gfCNCPoint5[2424] = {X 421.3630, Y 54.1078, Z -6.3333, A 0.000, B 0.000, C 0.000 }
gfCNCPoint5[2425] = {X 422.1821, Y 54.6225, Z -6.3333, A 0.000, B 0.000, C 0.000 }
gfCNCPoint5[2426] = {X 422.8661, Y 55.3065, Z -6.3333, A 0.000, B 0.000, C 0.000 }
gfCNCPoint5[2427] = {X 423.3808, Y 56.1256, Z -6.3333, A 0.000, B 0.000, C 0.000 }
gfCNCPoint5[2428] = {X 423.7003, Y 57.0387, Z -6.3333, A 0.000, B 0.000, C 0.000 }
gfCNCPoint5[2429] = {X 423.8086, Y 58.0000, Z -6.3333, A 0.000, B 0.000, C 0.000 }
gfCNCPoint5[2430] = {X 423.8086, Y 58.2318, Z -6.3333, A 0.000, B 0.000, C 0.000 }
gfCNCPoint5[2431] = {X 429.6116, Y 60.4927, Z -6.3333, A 0.000, B 0.000, C 0.000 }
gfCNCPoint5[2432] = {X 457.8582, Y 71.7001, Z -6.3333, A 0.000, B 0.000, C 0.000 }
gfCNCPoint5[2433] = {X 457.8604, Y 63.2123, Z -6.3333, A 0.000, B 0.000, C 0.000 }
gfCNCPoint5[2434] = {X 457.0088, Y 63.0032, Z -6.3333, A 0.000, B 0.000, C 0.000 }
gfCNCPoint5[2435] = {X 456.2169, Y 62.6263, Z -6.3333, A 0.000, B 0.000, C 0.000 }
gfCNCPoint5[2436] = {X 455.5175, Y 62.0974, Z -6.3333, A 0.000, B 0.000, C 0.000 }
gfCNCPoint5[2437] = {X 454.9393, Y 61.4381, Z -6.3333, A 0.000, B 0.000, C 0.000 }
gfCNCPoint5[2438] = {X 454.5062, Y 60.6756, Z -6.3333, A 0.000, B 0.000, C 0.000 }
gfCNCPoint5[2439] = {X 454.2360, Y 59.8414, Z -6.3333, A 0.000, B 0.000, C 0.000 }
gfCNCPoint5[2440] = {X 454.1398, Y 58.9697, Z -6.3333, A 0.000, B 0.000, C 0.000 }
gfCNCPoint5[2441] = {X 454.1396, Y 58.0000, Z -6.3333, A 0.000, B 0.000, C 0.000 }
gfCNCPoint5[2442] = {X 454.2479, Y 57.0387, Z -6.3333, A 0.000, B 0.000, C 0.000 }
gfCNCPoint5[2443] = {X 454.5674, Y 56.1256, Z -6.3333, A 0.000, B 0.000, C 0.000 }
gfCNCPoint5[2444] = {X 455.0821, Y 55.3065, Z -6.3333, A 0.000, B 0.000, C 0.000 }
gfCNCPoint5[2445] = {X 455.7661, Y 54.6225, Z -6.3333, A 0.000, B 0.000, C 0.000 }
gfCNCPoint5[2446] = {X 456.5852, Y 54.1078, Z -6.3333, A 0.000, B 0.000, C 0.000 }
gfCNCPoint5[2447] = {X 457.4983, Y 53.7883, Z -6.3333, A 0.000, B 0.000, C 0.000 }
gfCNCPoint5[2448] = {X 458.4596, Y 53.6800, Z -6.3333, A 0.000, B 0.000, C 0.000 }
gfCNCPoint5[2449] = {X 475.0000, Y 53.6800, Z -6.3333, A 0.000, B 0.000, C 0.000 }
gfCNCPoint5[2450] = {X 475.9613, Y 53.7883, Z -6.3333, A 0.000, B 0.000, C 0.000 }
gfCNCPoint5[2451] = {X 476.8744, Y 54.1078, Z -6.3333, A 0.000, B 0.000, C 0.000 }
gfCNCPoint5[2452] = {X 477.6935, Y 54.6225, Z -6.3333, A 0.000, B 0.000, C 0.000 }
gfCNCPoint5[2453] = {X 478.3775, Y 55.3065, Z -6.3333, A 0.000, B 0.000, C 0.000 }
gfCNCPoint5[2454] = {X 478.8922, Y 56.1256, Z -6.3333, A 0.000, B 0.000, C 0.000 }
gfCNCPoint5[2455] = {X 479.2117, Y 57.0387, Z -6.3333, A 0.000, B 0.000, C 0.000 }
gfCNCPoint5[2456] = {X 479.3200, Y 58.0000, Z -6.3333, A 0.000, B 0.000, C 0.000 }
gfCNCPoint5[2457] = {X 479.3200, Y 58.9342, Z -6.3333, A 0.000, B 0.000, C 0.000 }
gfCNCPoint5[2458] = {X 479.2300, Y 59.8114, Z -6.3333, A 0.000, B 0.000, C 0.000 }
gfCNCPoint5[2459] = {X 478.9637, Y 60.6520, Z -6.3333, A 0.000, B 0.000, C 0.000 }
gfCNCPoint5[2460] = {X 478.5324, Y 61.4210, Z -6.3333, A 0.000, B 0.000, C 0.000 }
gfCNCPoint5[2461] = {X 477.9538, Y 62.0864, Z -6.3333, A 0.000, B 0.000, C 0.000 }
gfCNCPoint5[2462] = {X 477.2523, Y 62.6205, Z -6.3333, A 0.000, B 0.000, C 0.000 }
gfCNCPoint5[2463] = {X 476.4568, Y 63.0010, Z -6.3333, A 0.000, B 0.000, C 0.000 }
gfCNCPoint5[2464] = {X 475.6007, Y 63.2121, Z -6.3333, A 0.000, B 0.000, C 0.000 }
gfCNCPoint5[2465] = {X 475.6012, Y 92.7676, Z -6.3333, A 0.000, B 0.000, C 0.000 }
gfCNCPoint5[2466] = {X 475.9931, Y 92.8655, Z -6.3333, A 0.000, B 0.000, C 0.000 }
gfCNCPoint5[2467] = {X 476.3796, Y 92.9832, Z -6.3333, A 0.000, B 0.000, C 0.000 }
gfCNCPoint5[2468] = {X 477.1933, Y 93.3521, Z -6.3333, A 0.000, B 0.000, C 0.000 }
gfCNCPoint5[2469] = {X 477.9133, Y 93.8812, Z -6.3333, A 0.000, B 0.000, C 0.000 }
gfCNCPoint5[2470] = {X 478.5083, Y 94.5477, Z -6.3333, A 0.000, B 0.000, C 0.000 }
gfCNCPoint5[2471] = {X 478.9526, Y 95.3228, Z -6.3333, A 0.000, B 0.000, C 0.000 }
gfCNCPoint5[2472] = {X 479.2272, Y 96.1731, Z -6.3333, A 0.000, B 0.000, C 0.000 }
gfCNCPoint5[2473] = {X 479.3200, Y 97.0617, Z -6.3333, A 0.000, B 0.000, C 0.000 }
gfCNCPoint5[2474] = {X 479.3200, Y 98.0000, Z -6.3333, A 0.000, B 0.000, C 0.000 }
gfCNCPoint5[2475] = {X 479.2117, Y 98.9613, Z -6.3333, A 0.000, B 0.000, C 0.000 }
gfCNCPoint5[2476] = {X 478.8922, Y 99.8744, Z -6.3333, A 0.000, B 0.000, C 0.000 }
gfCNCPoint5[2477] = {X 478.3775, Y 100.6935, Z -6.3333, A 0.000, B 0.000, C 0.000 }
gfCNCPoint5[2478] = {X 477.6935, Y 101.3775, Z -6.3333, A 0.000, B 0.000, C 0.000 }
gfCNCPoint5[2479] = {X 476.8744, Y 101.8922, Z -6.3333, A 0.000, B 0.000, C 0.000 }
gfCNCPoint5[2480] = {X 475.9613, Y 102.2117, Z -6.3333, A 0.000, B 0.000, C 0.000 }
gfCNCPoint5[2481] = {X 475.0000, Y 102.3200, Z -6.3333, A 0.000, B 0.000, C 0.000 }
gfCNCPoint5[2482] = {X 458.4596, Y 102.3200, Z -6.3333, A 0.000, B 0.000, C 0.000 }
gfCNCPoint5[2483] = {X 457.4983, Y 102.2117, Z -6.3333, A 0.000, B 0.000, C 0.000 }
gfCNCPoint5[2484] = {X 456.5852, Y 101.8922, Z -6.3333, A 0.000, B 0.000, C 0.000 }
gfCNCPoint5[2485] = {X 455.7661, Y 101.3775, Z -6.3333, A 0.000, B 0.000, C 0.000 }
gfCNCPoint5[2486] = {X 455.0821, Y 100.6935, Z -6.3333, A 0.000, B 0.000, C 0.000 }
gfCNCPoint5[2487] = {X 454.5674, Y 99.8744, Z -6.3333, A 0.000, B 0.000, C 0.000 }
gfCNCPoint5[2488] = {X 454.2479, Y 98.9613, Z -6.3333, A 0.000, B 0.000, C 0.000 }
gfCNCPoint5[2489] = {X 454.1396, Y 98.0000, Z -6.3333, A 0.000, B 0.000, C 0.000 }
gfCNCPoint5[2490] = {X 454.1396, Y 97.0659, Z -6.3333, A 0.000, B 0.000, C 0.000 }
gfCNCPoint5[2491] = {X 454.2295, Y 96.1891, Z -6.3333, A 0.000, B 0.000, C 0.000 }
gfCNCPoint5[2492] = {X 454.4955, Y 95.3488, Z -6.3333, A 0.000, B 0.000, C 0.000 }
gfCNCPoint5[2493] = {X 454.9265, Y 94.5800, Z -6.3333, A 0.000, B 0.000, C 0.000 }
gfCNCPoint5[2494] = {X 455.5046, Y 93.9147, Z -6.3333, A 0.000, B 0.000, C 0.000 }
gfCNCPoint5[2495] = {X 456.2057, Y 93.3805, Z -6.3333, A 0.000, B 0.000, C 0.000 }
gfCNCPoint5[2496] = {X 457.0006, Y 92.9998, Z -6.3333, A 0.000, B 0.000, C 0.000 }
gfCNCPoint5[2497] = {X 457.8563, Y 92.7883, Z -6.3333, A 0.000, B 0.000, C 0.000 }
gfCNCPoint5[2498] = {X 457.8563, Y 85.5950, Z -6.3333, A 0.000, B 0.000, C 0.000 }
gfCNCPoint5[2499] = {X 444.8598, Y 80.5003, Z -6.3333, A 0.000, B 0.000, C 0.000 }
gfCNCPoint5[2500] = {X 420.0239, Y 96.5884, Z -6.3333, A 0.000, B 0.000, C 0.000 }
gfCNCPoint5[2501] = {X 420.0267, Y 97.0650, Z -6.3333, A 0.000, B 0.000, C 0.000 }
gfCNCPoint5[2502] = {X 420.0267, Y 98.0000, Z -6.3333, A 0.000, B 0.000, C 0.000 }
gfCNCPoint5[2503] = {X 419.9184, Y 98.9613, Z -6.3333, A 0.000, B 0.000, C 0.000 }
gfCNCPoint5[2504] = {X 419.5989, Y 99.8744, Z -6.3333, A 0.000, B 0.000, C 0.000 }
gfCNCPoint5[2505] = {X 419.0842, Y 100.6935, Z -6.3333, A 0.000, B 0.000, C 0.000 }
gfCNCPoint5[2506] = {X 418.4002, Y 101.3775, Z -6.3333, A 0.000, B 0.000, C 0.000 }
gfCNCPoint5[2507] = {X 417.5811, Y 101.8922, Z -6.3333, A 0.000, B 0.000, C 0.000 }
gfCNCPoint5[2508] = {X 416.6680, Y 102.2117, Z -6.3333, A 0.000, B 0.000, C 0.000 }
gfCNCPoint5[2509] = {X 415.7067, Y 102.3200, Z -6.3333, A 0.000, B 0.000, C 0.000 }
gfCNCPoint5[2510] = {X 396.4059, Y 102.3200, Z -6.3333, A 0.000, B 0.000, C 0.000 }
gfCNCPoint5[2511] = {X 395.4447, Y 102.2117, Z -6.3333, A 0.000, B 0.000, C 0.000 }
gfCNCPoint5[2512] = {X 394.5316, Y 101.8922, Z -6.3333, A 0.000, B 0.000, C 0.000 }
gfCNCPoint5[2513] = {X 393.7125, Y 101.3775, Z -6.3333, A 0.000, B 0.000, C 0.000 }
gfCNCPoint5[2514] = {X 393.0284, Y 100.6935, Z -6.3333, A 0.000, B 0.000, C 0.000 }
gfCNCPoint5[2515] = {X 392.5138, Y 99.8744, Z -6.3333, A 0.000, B 0.000, C 0.000 }
gfCNCPoint5[2516] = {X 392.1943, Y 98.9613, Z -6.3333, A 0.000, B 0.000, C 0.000 }
gfCNCPoint5[2517] = {X 392.0859, Y 98.0000, Z -6.3333, A 0.000, B 0.000, C 0.000 }
gfCNCPoint5[2518] = {X 392.0859, Y 97.0659, Z -6.3333, A 0.000, B 0.000, C 0.000 }
gfCNCPoint5[2519] = {X 392.1944, Y 96.1042, Z -6.3333, A 0.000, B 0.000, C 0.000 }
gfCNCPoint5[2520] = {X 392.5142, Y 95.1907, Z -6.3333, A 0.000, B 0.000, C 0.000 }
gfCNCPoint5[2521] = {X 393.0293, Y 94.3714, Z -6.3333, A 0.000, B 0.000, C 0.000 }
gfCNCPoint5[2522] = {X 393.7139, Y 93.6872, Z -6.3333, A 0.000, B 0.000, C 0.000 }
gfCNCPoint5[2523] = {X 394.5337, Y 93.1727, Z -6.3333, A 0.000, B 0.000, C 0.000 }
gfCNCPoint5[2524] = {X 395.4474, Y 92.8536, Z -6.3333, A 0.000, B 0.000, C 0.000 }
gfCNCPoint5[2525] = {X 396.4092, Y 92.7459, Z -6.3333, A 0.000, B 0.000, C 0.000 }
gfCNCPoint5[2526] = {X 397.3530, Y 92.7029, Z -6.3333, A 0.000, B 0.000, C 0.000 }
gfCNCPoint5[2527] = {X 398.2934, Y 92.6137, Z -6.3333, A 0.000, B 0.000, C 0.000 }
gfCNCPoint5[2528] = {X 398.9443, Y 92.4557, Z -6.3333, A 0.000, B 0.000, C 0.000 }
gfCNCPoint5[2529] = {X 399.5438, Y 92.1569, Z -6.3333, A 0.000, B 0.000, C 0.000 }
gfCNCPoint5[2530] = {X 413.7988, Y 83.0282, Z -6.3333, A 0.000, B 0.000, C 0.000 }
gfCNCPoint5[2531] = {X 411.6417, Y 79.6597, Z -6.3333, A 0.000, B 0.000, C 0.000 }
gfCNCPoint5[2532] = {X 413.8419, Y 83.0956, Z -6.3333, A 0.000, B 0.000, C 0.000 }
gfCNCPoint5[2533] = {X 428.2290, Y 73.8824, Z -6.3333, A 0.000, B 0.000, C 0.000 }
gfCNCPoint5[2534] = {X 403.7848, Y 64.2921, Z -6.3333, A 0.000, B 0.000, C 0.000 }
gfCNCPoint5[2535] = {X 402.0800, Y 63.7277, Z -6.3333, A 0.000, B 0.000, C 0.000 }
gfCNCPoint5[2536] = {X 400.3236, Y 63.3536, Z -6.3333, A 0.000, B 0.000, C 0.000 }
gfCNCPoint5[2537] = {X 398.5368, Y 63.1740, Z -6.3333, A 0.000, B 0.000, C 0.000 }
gfCNCPoint5[2538] = {X 397.6016, Y 63.0649, Z -6.3333, A 0.000, B 0.000, C 0.000 }
gfCNCPoint5[2539] = {X 396.7136, Y 62.7520, Z -6.3333, A 0.000, B 0.000, C 0.000 }
gfCNCPoint5[2540] = {X 395.9166, Y 62.2510, Z -6.3333, A 0.000, B 0.000, C 0.000 }
gfCNCPoint5[2541] = {X 395.2497, Y 61.5864, Z -6.3333, A 0.000, B 0.000, C 0.000 }
gfCNCPoint5[2542] = {X 394.7460, Y 60.7910, Z -6.3333, A 0.000, B 0.000, C 0.000 }
gfCNCPoint5[2543] = {X 394.4302, Y 59.9040, Z -6.3333, A 0.000, B 0.000, C 0.000 }
gfCNCPoint5[2544] = {X 394.3179, Y 58.9693, Z -6.3333, A 0.000, B 0.000, C 0.000 }
gfCNCPoint5[2545] = {X 394.3177, Y 58.0000, Z -6.3333, A 0.000, B 0.000, C 0.000 }
gfCNCPoint5[2546] = {X 394.4240, Y 57.0565, Z -6.3333, A 0.000, B 0.000, C 0.000 }
gfCNCPoint5[2547] = {X 394.7376, Y 56.1603, Z -6.3333, A 0.000, B 0.000, C 0.000 }
gfCNCPoint5[2548] = {X 395.2428, Y 55.3564, Z -6.3333, A 0.000, B 0.000, C 0.000 }
gfCNCPoint5[2549] = {X 395.9141, Y 54.6850, Z -6.3333, A 0.000, B 0.000, C 0.000 }
gfCNCPoint5[2550] = {X 396.7181, Y 54.1799, Z -6.3333, A 0.000, B 0.000, C 0.000 }
gfCNCPoint5[2551] = {X 397.6142, Y 53.8663, Z -6.3333, A 0.000, B 0.000, C 0.000 }
gfCNCPoint5[2552] = {X 398.5577, Y 53.7600, Z -6.3333, A 0.000, B 0.000, C 0.000 }
gfCNCPoint5[2553] = {X 419.4886, Y 53.7600, Z -6.3333, A 0.000, B 0.000, C 0.000 }
gfCNCPoint5[2554] = {X 420.4321, Y 53.8663, Z -6.3333, A 0.000, B 0.000, C 0.000 }
gfCNCPoint5[2555] = {X 421.3283, Y 54.1799, Z -6.3333, A 0.000, B 0.000, C 0.000 }
gfCNCPoint5[2556] = {X 422.1322, Y 54.6850, Z -6.3333, A 0.000, B 0.000, C 0.000 }
gfCNCPoint5[2557] = {X 422.8036, Y 55.3564, Z -6.3333, A 0.000, B 0.000, C 0.000 }
gfCNCPoint5[2558] = {X 423.3087, Y 56.1603, Z -6.3333, A 0.000, B 0.000, C 0.000 }
gfCNCPoint5[2559] = {X 423.6223, Y 57.0565, Z -6.3333, A 0.000, B 0.000, C 0.000 }
gfCNCPoint5[2560] = {X 423.7286, Y 58.0000, Z -6.3333, A 0.000, B 0.000, C 0.000 }
gfCNCPoint5[2561] = {X 423.7286, Y 58.2864, Z -6.3333, A 0.000, B 0.000, C 0.000 }
gfCNCPoint5[2562] = {X 429.5823, Y 60.5672, Z -6.3333, A 0.000, B 0.000, C 0.000 }
gfCNCPoint5[2563] = {X 457.9382, Y 71.8179, Z -6.3333, A 0.000, B 0.000, C 0.000 }
gfCNCPoint5[2564] = {X 457.9404, Y 63.1422, Z -6.3333, A 0.000, B 0.000, C 0.000 }
gfCNCPoint5[2565] = {X 457.0919, Y 62.9474, Z -6.3333, A 0.000, B 0.000, C 0.000 }
gfCNCPoint5[2566] = {X 456.3011, Y 62.5835, Z -6.3333, A 0.000, B 0.000, C 0.000 }
gfCNCPoint5[2567] = {X 455.6012, Y 62.0657, Z -6.3333, A 0.000, B 0.000, C 0.000 }
gfCNCPoint5[2568] = {X 455.0219, Y 61.4159, Z -6.3333, A 0.000, B 0.000, C 0.000 }
gfCNCPoint5[2569] = {X 454.5875, Y 60.6615, Z -6.3333, A 0.000, B 0.000, C 0.000 }
gfCNCPoint5[2570] = {X 454.3163, Y 59.8343, Z -6.3333, A 0.000, B 0.000, C 0.000 }
gfCNCPoint5[2571] = {X 454.2197, Y 58.9691, Z -6.3333, A 0.000, B 0.000, C 0.000 }
gfCNCPoint5[2572] = {X 454.2196, Y 58.0000, Z -6.3333, A 0.000, B 0.000, C 0.000 }
gfCNCPoint5[2573] = {X 454.3259, Y 57.0565, Z -6.3333, A 0.000, B 0.000, C 0.000 }
gfCNCPoint5[2574] = {X 454.6395, Y 56.1603, Z -6.3333, A 0.000, B 0.000, C 0.000 }
gfCNCPoint5[2575] = {X 455.1446, Y 55.3564, Z -6.3333, A 0.000, B 0.000, C 0.000 }
gfCNCPoint5[2576] = {X 455.8160, Y 54.6850, Z -6.3333, A 0.000, B 0.000, C 0.000 }
gfCNCPoint5[2577] = {X 456.6199, Y 54.1799, Z -6.3333, A 0.000, B 0.000, C 0.000 }
gfCNCPoint5[2578] = {X 457.5161, Y 53.8663, Z -6.3333, A 0.000, B 0.000, C 0.000 }
gfCNCPoint5[2579] = {X 458.4596, Y 53.7600, Z -6.3333, A 0.000, B 0.000, C 0.000 }
gfCNCPoint5[2580] = {X 475.0000, Y 53.7600, Z -6.3333, A 0.000, B 0.000, C 0.000 }
gfCNCPoint5[2581] = {X 475.9435, Y 53.8663, Z -6.3333, A 0.000, B 0.000, C 0.000 }
gfCNCPoint5[2582] = {X 476.8397, Y 54.1799, Z -6.3333, A 0.000, B 0.000, C 0.000 }
gfCNCPoint5[2583] = {X 477.6436, Y 54.6850, Z -6.3333, A 0.000, B 0.000, C 0.000 }
gfCNCPoint5[2584] = {X 478.3150, Y 55.3564, Z -6.3333, A 0.000, B 0.000, C 0.000 }
gfCNCPoint5[2585] = {X 478.8201, Y 56.1603, Z -6.3333, A 0.000, B 0.000, C 0.000 }
gfCNCPoint5[2586] = {X 479.1337, Y 57.0565, Z -6.3333, A 0.000, B 0.000, C 0.000 }
gfCNCPoint5[2587] = {X 479.2400, Y 58.0000, Z -6.3333, A 0.000, B 0.000, C 0.000 }
gfCNCPoint5[2588] = {X 479.2400, Y 58.9342, Z -6.3333, A 0.000, B 0.000, C 0.000 }
gfCNCPoint5[2589] = {X 479.1496, Y 59.8048, Z -6.3333, A 0.000, B 0.000, C 0.000 }
gfCNCPoint5[2590] = {X 478.8824, Y 60.6383, Z -6.3333, A 0.000, B 0.000, C 0.000 }
gfCNCPoint5[2591] = {X 478.4497, Y 61.3992, Z -6.3333, A 0.000, B 0.000, C 0.000 }
gfCNCPoint5[2592] = {X 477.8700, Y 62.0550, Z -6.3333, A 0.000, B 0.000, C 0.000 }
gfCNCPoint5[2593] = {X 477.1680, Y 62.5778, Z -6.3333, A 0.000, B 0.000, C 0.000 }
gfCNCPoint5[2594] = {X 476.3737, Y 62.9454, Z -6.3333, A 0.000, B 0.000, C 0.000 }
gfCNCPoint5[2595] = {X 475.5207, Y 63.1420, Z -6.3333, A 0.000, B 0.000, C 0.000 }
gfCNCPoint5[2596] = {X 475.5212, Y 92.8321, Z -6.3333, A 0.000, B 0.000, C 0.000 }
gfCNCPoint5[2597] = {X 475.9409, Y 92.9341, Z -6.3333, A 0.000, B 0.000, C 0.000 }
gfCNCPoint5[2598] = {X 476.3543, Y 93.0591, Z -6.3333, A 0.000, B 0.000, C 0.000 }
gfCNCPoint5[2599] = {X 477.1529, Y 93.4211, Z -6.3333, A 0.000, B 0.000, C 0.000 }
gfCNCPoint5[2600] = {X 477.8594, Y 93.9404, Z -6.3333, A 0.000, B 0.000, C 0.000 }
gfCNCPoint5[2601] = {X 478.4434, Y 94.5945, Z -6.3333, A 0.000, B 0.000, C 0.000 }
gfCNCPoint5[2602] = {X 478.8795, Y 95.3552, Z -6.3333, A 0.000, B 0.000, C 0.000 }
gfCNCPoint5[2603] = {X 479.1489, Y 96.1896, Z -6.3333, A 0.000, B 0.000, C 0.000 }
gfCNCPoint5[2604] = {X 479.2400, Y 97.0617, Z -6.3333, A 0.000, B 0.000, C 0.000 }
gfCNCPoint5[2605] = {X 479.2400, Y 98.0000, Z -6.3333, A 0.000, B 0.000, C 0.000 }
gfCNCPoint5[2606] = {X 479.1337, Y 98.9435, Z -6.3333, A 0.000, B 0.000, C 0.000 }
gfCNCPoint5[2607] = {X 478.8201, Y 99.8397, Z -6.3333, A 0.000, B 0.000, C 0.000 }
gfCNCPoint5[2608] = {X 478.3150, Y 100.6436, Z -6.3333, A 0.000, B 0.000, C 0.000 }
gfCNCPoint5[2609] = {X 477.6436, Y 101.3150, Z -6.3333, A 0.000, B 0.000, C 0.000 }
gfCNCPoint5[2610] = {X 476.8397, Y 101.8201, Z -6.3333, A 0.000, B 0.000, C 0.000 }
gfCNCPoint5[2611] = {X 475.9435, Y 102.1337, Z -6.3333, A 0.000, B 0.000, C 0.000 }
gfCNCPoint5[2612] = {X 475.0000, Y 102.2400, Z -6.3333, A 0.000, B 0.000, C 0.000 }
gfCNCPoint5[2613] = {X 458.4596, Y 102.2400, Z -6.3333, A 0.000, B 0.000, C 0.000 }
gfCNCPoint5[2614] = {X 457.5161, Y 102.1337, Z -6.3333, A 0.000, B 0.000, C 0.000 }
gfCNCPoint5[2615] = {X 456.6199, Y 101.8201, Z -6.3333, A 0.000, B 0.000, C 0.000 }
gfCNCPoint5[2616] = {X 455.8160, Y 101.3150, Z -6.3333, A 0.000, B 0.000, C 0.000 }
gfCNCPoint5[2617] = {X 455.1446, Y 100.6436, Z -6.3333, A 0.000, B 0.000, C 0.000 }
gfCNCPoint5[2618] = {X 454.6395, Y 99.8397, Z -6.3333, A 0.000, B 0.000, C 0.000 }
gfCNCPoint5[2619] = {X 454.3259, Y 98.9435, Z -6.3333, A 0.000, B 0.000, C 0.000 }
gfCNCPoint5[2620] = {X 454.2196, Y 98.0000, Z -6.3333, A 0.000, B 0.000, C 0.000 }
gfCNCPoint5[2621] = {X 454.2196, Y 97.0659, Z -6.3333, A 0.000, B 0.000, C 0.000 }
gfCNCPoint5[2622] = {X 454.3099, Y 96.1957, Z -6.3333, A 0.000, B 0.000, C 0.000 }
gfCNCPoint5[2623] = {X 454.5769, Y 95.3624, Z -6.3333, A 0.000, B 0.000, C 0.000 }
gfCNCPoint5[2624] = {X 455.0092, Y 94.6018, Z -6.3333, A 0.000, B 0.000, C 0.000 }
gfCNCPoint5[2625] = {X 455.5884, Y 93.9460, Z -6.3333, A 0.000, B 0.000, C 0.000 }
gfCNCPoint5[2626] = {X 456.2899, Y 93.4231, Z -6.3333, A 0.000, B 0.000, C 0.000 }
gfCNCPoint5[2627] = {X 457.0838, Y 93.0553, Z -6.3333, A 0.000, B 0.000, C 0.000 }
gfCNCPoint5[2628] = {X 457.9363, Y 92.8584, Z -6.3333, A 0.000, B 0.000, C 0.000 }
gfCNCPoint5[2629] = {X 457.9363, Y 85.5404, Z -6.3333, A 0.000, B 0.000, C 0.000 }
gfCNCPoint5[2630] = {X 444.8508, Y 80.4109, Z -6.3333, A 0.000, B 0.000, C 0.000 }
gfCNCPoint5[2631] = {X 419.9437, Y 96.5451, Z -6.3333, A 0.000, B 0.000, C 0.000 }
gfCNCPoint5[2632] = {X 419.9467, Y 97.0652, Z -6.3333, A 0.000, B 0.000, C 0.000 }
gfCNCPoint5[2633] = {X 419.9467, Y 98.0000, Z -6.3333, A 0.000, B 0.000, C 0.000 }
gfCNCPoint5[2634] = {X 419.8404, Y 98.9435, Z -6.3333, A 0.000, B 0.000, C 0.000 }
gfCNCPoint5[2635] = {X 419.5268, Y 99.8397, Z -6.3333, A 0.000, B 0.000, C 0.000 }
gfCNCPoint5[2636] = {X 419.0217, Y 100.6436, Z -6.3333, A 0.000, B 0.000, C 0.000 }
gfCNCPoint5[2637] = {X 418.3503, Y 101.3150, Z -6.3333, A 0.000, B 0.000, C 0.000 }
gfCNCPoint5[2638] = {X 417.5464, Y 101.8201, Z -6.3333, A 0.000, B 0.000, C 0.000 }
gfCNCPoint5[2639] = {X 416.6502, Y 102.1337, Z -6.3333, A 0.000, B 0.000, C 0.000 }
gfCNCPoint5[2640] = {X 415.7067, Y 102.2400, Z -6.3333, A 0.000, B 0.000, C 0.000 }
gfCNCPoint5[2641] = {X 396.4059, Y 102.2400, Z -6.3333, A 0.000, B 0.000, C 0.000 }
gfCNCPoint5[2642] = {X 395.4625, Y 102.1337, Z -6.3333, A 0.000, B 0.000, C 0.000 }
gfCNCPoint5[2643] = {X 394.5663, Y 101.8201, Z -6.3333, A 0.000, B 0.000, C 0.000 }
gfCNCPoint5[2644] = {X 393.7624, Y 101.3150, Z -6.3333, A 0.000, B 0.000, C 0.000 }
gfCNCPoint5[2645] = {X 393.0910, Y 100.6436, Z -6.3333, A 0.000, B 0.000, C 0.000 }
gfCNCPoint5[2646] = {X 392.5858, Y 99.8397, Z -6.3333, A 0.000, B 0.000, C 0.000 }
gfCNCPoint5[2647] = {X 392.2723, Y 98.9435, Z -6.3333, A 0.000, B 0.000, C 0.000 }
gfCNCPoint5[2648] = {X 392.1659, Y 98.0000, Z -6.3333, A 0.000, B 0.000, C 0.000 }
gfCNCPoint5[2649] = {X 392.1659, Y 97.0659, Z -6.3333, A 0.000, B 0.000, C 0.000 }
gfCNCPoint5[2650] = {X 392.2724, Y 96.1219, Z -6.3333, A 0.000, B 0.000, C 0.000 }
gfCNCPoint5[2651] = {X 392.5864, Y 95.2252, Z -6.3333, A 0.000, B 0.000, C 0.000 }
gfCNCPoint5[2652] = {X 393.0921, Y 94.4210, Z -6.3333, A 0.000, B 0.000, C 0.000 }
gfCNCPoint5[2653] = {X 393.7642, Y 93.7495, Z -6.3333, A 0.000, B 0.000, C 0.000 }
gfCNCPoint5[2654] = {X 394.5689, Y 93.2446, Z -6.3333, A 0.000, B 0.000, C 0.000 }
gfCNCPoint5[2655] = {X 395.4659, Y 92.9315, Z -6.3333, A 0.000, B 0.000, C 0.000 }
gfCNCPoint5[2656] = {X 396.4101, Y 92.8259, Z -6.3333, A 0.000, B 0.000, C 0.000 }
gfCNCPoint5[2657] = {X 397.3583, Y 92.7828, Z -6.3333, A 0.000, B 0.000, C 0.000 }
gfCNCPoint5[2658] = {X 398.3033, Y 92.6930, Z -6.3333, A 0.000, B 0.000, C 0.000 }
gfCNCPoint5[2659] = {X 398.9717, Y 92.5309, Z -6.3333, A 0.000, B 0.000, C 0.000 }
gfCNCPoint5[2660] = {X 399.5872, Y 92.2241, Z -6.3333, A 0.000, B 0.000, C 0.000 }
gfCNCPoint5[2661] = {X 413.8419, Y 83.0956, Z -6.3333, A 0.000, B 0.000, C 0.000 }
gfCNCPoint5[2662] = {X 411.6848, Y 79.7271, Z -6.3333, A 0.000, B 0.000, C 0.000 }
gfCNCPoint5[2663] = {X 413.8851, Y 83.1630, Z -6.3333, A 0.000, B 0.000, C 0.000 }
gfCNCPoint5[2664] = {X 428.4042, Y 73.8652, Z -6.3333, A 0.000, B 0.000, C 0.000 }
gfCNCPoint5[2665] = {X 403.8141, Y 64.2176, Z -6.3333, A 0.000, B 0.000, C 0.000 }
gfCNCPoint5[2666] = {X 402.1004, Y 63.6504, Z -6.3333, A 0.000, B 0.000, C 0.000 }
gfCNCPoint5[2667] = {X 400.3349, Y 63.2744, Z -6.3333, A 0.000, B 0.000, C 0.000 }
gfCNCPoint5[2668] = {X 398.5388, Y 63.0940, Z -6.3333, A 0.000, B 0.000, C 0.000 }
gfCNCPoint5[2669] = {X 397.6210, Y 62.9872, Z -6.3333, A 0.000, B 0.000, C 0.000 }
gfCNCPoint5[2670] = {X 396.7495, Y 62.6805, Z -6.3333, A 0.000, B 0.000, C 0.000 }
gfCNCPoint5[2671] = {X 395.9671, Y 62.1890, Z -6.3333, A 0.000, B 0.000, C 0.000 }
gfCNCPoint5[2672] = {X 395.3126, Y 61.5369, Z -6.3333, A 0.000, B 0.000, C 0.000 }
gfCNCPoint5[2673] = {X 394.8181, Y 60.7564, Z -6.3333, A 0.000, B 0.000, C 0.000 }
gfCNCPoint5[2674] = {X 394.5081, Y 59.8860, Z -6.3333, A 0.000, B 0.000, C 0.000 }
gfCNCPoint5[2675] = {X 394.3979, Y 58.9686, Z -6.3333, A 0.000, B 0.000, C 0.000 }
gfCNCPoint5[2676] = {X 394.3977, Y 58.0000, Z -6.3333, A 0.000, B 0.000, C 0.000 }
gfCNCPoint5[2677] = {X 394.5020, Y 57.0743, Z -6.3333, A 0.000, B 0.000, C 0.000 }
gfCNCPoint5[2678] = {X 394.8097, Y 56.1950, Z -6.3333, A 0.000, B 0.000, C 0.000 }
gfCNCPoint5[2679] = {X 395.3053, Y 55.4063, Z -6.3333, A 0.000, B 0.000, C 0.000 }
gfCNCPoint5[2680] = {X 395.9640, Y 54.7476, Z -6.3333, A 0.000, B 0.000, C 0.000 }
gfCNCPoint5[2681] = {X 396.7528, Y 54.2520, Z -6.3333, A 0.000, B 0.000, C 0.000 }
gfCNCPoint5[2682] = {X 397.6320, Y 53.9443, Z -6.3333, A 0.000, B 0.000, C 0.000 }
gfCNCPoint5[2683] = {X 398.5577, Y 53.8400, Z -6.3333, A 0.000, B 0.000, C 0.000 }
gfCNCPoint5[2684] = {X 419.4886, Y 53.8400, Z -6.3333, A 0.000, B 0.000, C 0.000 }
gfCNCPoint5[2685] = {X 420.4143, Y 53.9443, Z -6.3333, A 0.000, B 0.000, C 0.000 }
gfCNCPoint5[2686] = {X 421.2936, Y 54.2520, Z -6.3333, A 0.000, B 0.000, C 0.000 }
gfCNCPoint5[2687] = {X 422.0823, Y 54.7476, Z -6.3333, A 0.000, B 0.000, C 0.000 }
gfCNCPoint5[2688] = {X 422.7410, Y 55.4063, Z -6.3333, A 0.000, B 0.000, C 0.000 }
gfCNCPoint5[2689] = {X 423.2366, Y 56.1950, Z -6.3333, A 0.000, B 0.000, C 0.000 }
gfCNCPoint5[2690] = {X 423.5443, Y 57.0743, Z -6.3333, A 0.000, B 0.000, C 0.000 }
gfCNCPoint5[2691] = {X 423.6486, Y 58.0000, Z -6.3333, A 0.000, B 0.000, C 0.000 }
gfCNCPoint5[2692] = {X 423.6486, Y 58.3411, Z -6.3333, A 0.000, B 0.000, C 0.000 }
gfCNCPoint5[2693] = {X 429.5530, Y 60.6416, Z -6.3333, A 0.000, B 0.000, C 0.000 }
gfCNCPoint5[2694] = {X 458.0182, Y 71.9357, Z -6.3333, A 0.000, B 0.000, C 0.000 }
gfCNCPoint5[2695] = {X 458.0204, Y 63.0708, Z -6.3333, A 0.000, B 0.000, C 0.000 }
gfCNCPoint5[2696] = {X 457.9179, Y 63.0586, Z -6.3333, A 0.000, B 0.000, C 0.000 }
gfCNCPoint5[2697] = {X 457.8157, Y 63.0439, Z -6.3333, A 0.000, B 0.000, C 0.000 }
gfCNCPoint5[2698] = {X 456.8783, Y 62.7818, Z -6.3333, A 0.000, B 0.000, C 0.000 }
gfCNCPoint5[2699] = {X 456.0274, Y 62.3090, Z -6.3333, A 0.000, B 0.000, C 0.000 }
gfCNCPoint5[2700] = {X 455.3098, Y 61.6514, Z -6.3333, A 0.000, B 0.000, C 0.000 }
gfCNCPoint5[2701] = {X 454.7645, Y 60.8451, Z -6.3333, A 0.000, B 0.000, C 0.000 }
gfCNCPoint5[2702] = {X 454.4216, Y 59.9341, Z -6.3333, A 0.000, B 0.000, C 0.000 }
gfCNCPoint5[2703] = {X 454.2997, Y 58.9684, Z -6.3333, A 0.000, B 0.000, C 0.000 }
gfCNCPoint5[2704] = {X 454.2996, Y 58.0000, Z -6.3333, A 0.000, B 0.000, C 0.000 }
gfCNCPoint5[2705] = {X 454.4039, Y 57.0743, Z -6.3333, A 0.000, B 0.000, C 0.000 }
gfCNCPoint5[2706] = {X 454.7116, Y 56.1950, Z -6.3333, A 0.000, B 0.000, C 0.000 }
gfCNCPoint5[2707] = {X 455.2072, Y 55.4063, Z -6.3333, A 0.000, B 0.000, C 0.000 }
gfCNCPoint5[2708] = {X 455.8659, Y 54.7476, Z -6.3333, A 0.000, B 0.000, C 0.000 }
gfCNCPoint5[2709] = {X 456.6546, Y 54.2520, Z -6.3333, A 0.000, B 0.000, C 0.000 }
gfCNCPoint5[2710] = {X 457.5339, Y 53.9443, Z -6.3333, A 0.000, B 0.000, C 0.000 }
gfCNCPoint5[2711] = {X 458.4596, Y 53.8400, Z -6.3333, A 0.000, B 0.000, C 0.000 }
gfCNCPoint5[2712] = {X 475.0000, Y 53.8400, Z -6.3333, A 0.000, B 0.000, C 0.000 }
gfCNCPoint5[2713] = {X 475.9257, Y 53.9443, Z -6.3333, A 0.000, B 0.000, C 0.000 }
gfCNCPoint5[2714] = {X 476.8050, Y 54.2520, Z -6.3333, A 0.000, B 0.000, C 0.000 }
gfCNCPoint5[2715] = {X 477.5937, Y 54.7476, Z -6.3333, A 0.000, B 0.000, C 0.000 }
gfCNCPoint5[2716] = {X 478.2524, Y 55.4063, Z -6.3333, A 0.000, B 0.000, C 0.000 }
gfCNCPoint5[2717] = {X 478.7480, Y 56.1950, Z -6.3333, A 0.000, B 0.000, C 0.000 }
gfCNCPoint5[2718] = {X 479.0557, Y 57.0743, Z -6.3333, A 0.000, B 0.000, C 0.000 }
gfCNCPoint5[2719] = {X 479.1600, Y 58.0000, Z -6.3333, A 0.000, B 0.000, C 0.000 }
gfCNCPoint5[2720] = {X 479.1600, Y 58.9342, Z -6.3333, A 0.000, B 0.000, C 0.000 }
gfCNCPoint5[2721] = {X 479.0692, Y 59.7983, Z -6.3333, A 0.000, B 0.000, C 0.000 }
gfCNCPoint5[2722] = {X 478.8010, Y 60.6246, Z -6.3333, A 0.000, B 0.000, C 0.000 }
gfCNCPoint5[2723] = {X 478.3669, Y 61.3773, Z -6.3333, A 0.000, B 0.000, C 0.000 }
gfCNCPoint5[2724] = {X 477.7860, Y 62.0233, Z -6.3333, A 0.000, B 0.000, C 0.000 }
gfCNCPoint5[2725] = {X 477.0836, Y 62.5346, Z -6.3333, A 0.000, B 0.000, C 0.000 }
gfCNCPoint5[2726] = {X 476.2903, Y 62.8889, Z -6.3333, A 0.000, B 0.000, C 0.000 }
gfCNCPoint5[2727] = {X 475.4407, Y 63.0707, Z -6.3333, A 0.000, B 0.000, C 0.000 }
gfCNCPoint5[2728] = {X 475.4412, Y 92.8970, Z -6.3333, A 0.000, B 0.000, C 0.000 }
gfCNCPoint5[2729] = {X 475.8887, Y 93.0028, Z -6.3333, A 0.000, B 0.000, C 0.000 }
gfCNCPoint5[2730] = {X 476.3290, Y 93.1350, Z -6.3333, A 0.000, B 0.000, C 0.000 }
gfCNCPoint5[2731] = {X 477.1125, Y 93.4902, Z -6.3333, A 0.000, B 0.000, C 0.000 }
gfCNCPoint5[2732] = {X 477.8056, Y 93.9996, Z -6.3333, A 0.000, B 0.000, C 0.000 }
gfCNCPoint5[2733] = {X 478.3785, Y 94.6413, Z -6.3333, A 0.000, B 0.000, C 0.000 }
gfCNCPoint5[2734] = {X 478.8063, Y 95.3876, Z -6.3333, A 0.000, B 0.000, C 0.000 }
gfCNCPoint5[2735] = {X 479.0706, Y 96.2061, Z -6.3333, A 0.000, B 0.000, C 0.000 }
gfCNCPoint5[2736] = {X 479.1600, Y 97.0617, Z -6.3333, A 0.000, B 0.000, C 0.000 }
gfCNCPoint5[2737] = {X 479.1600, Y 98.0000, Z -6.3333, A 0.000, B 0.000, C 0.000 }
gfCNCPoint5[2738] = {X 479.0557, Y 98.9257, Z -6.3333, A 0.000, B 0.000, C 0.000 }
gfCNCPoint5[2739] = {X 478.7480, Y 99.8050, Z -6.3333, A 0.000, B 0.000, C 0.000 }
gfCNCPoint5[2740] = {X 478.2524, Y 100.5937, Z -6.3333, A 0.000, B 0.000, C 0.000 }
gfCNCPoint5[2741] = {X 477.5937, Y 101.2524, Z -6.3333, A 0.000, B 0.000, C 0.000 }
gfCNCPoint5[2742] = {X 476.8050, Y 101.7480, Z -6.3333, A 0.000, B 0.000, C 0.000 }
gfCNCPoint5[2743] = {X 475.9257, Y 102.0557, Z -6.3333, A 0.000, B 0.000, C 0.000 }
gfCNCPoint5[2744] = {X 475.0000, Y 102.1600, Z -6.3333, A 0.000, B 0.000, C 0.000 }
gfCNCPoint5[2745] = {X 458.4596, Y 102.1600, Z -6.3333, A 0.000, B 0.000, C 0.000 }
gfCNCPoint5[2746] = {X 457.5339, Y 102.0557, Z -6.3333, A 0.000, B 0.000, C 0.000 }
gfCNCPoint5[2747] = {X 456.6546, Y 101.7480, Z -6.3333, A 0.000, B 0.000, C 0.000 }
gfCNCPoint5[2748] = {X 455.8659, Y 101.2524, Z -6.3333, A 0.000, B 0.000, C 0.000 }
gfCNCPoint5[2749] = {X 455.2072, Y 100.5937, Z -6.3333, A 0.000, B 0.000, C 0.000 }
gfCNCPoint5[2750] = {X 454.7116, Y 99.8050, Z -6.3333, A 0.000, B 0.000, C 0.000 }
gfCNCPoint5[2751] = {X 454.4039, Y 98.9257, Z -6.3333, A 0.000, B 0.000, C 0.000 }
gfCNCPoint5[2752] = {X 454.2996, Y 98.0000, Z -6.3333, A 0.000, B 0.000, C 0.000 }
gfCNCPoint5[2753] = {X 454.2996, Y 97.0659, Z -6.3333, A 0.000, B 0.000, C 0.000 }
gfCNCPoint5[2754] = {X 454.3903, Y 96.2022, Z -6.3333, A 0.000, B 0.000, C 0.000 }
gfCNCPoint5[2755] = {X 454.6583, Y 95.3761, Z -6.3333, A 0.000, B 0.000, C 0.000 }
gfCNCPoint5[2756] = {X 455.0920, Y 94.6237, Z -6.3333, A 0.000, B 0.000, C 0.000 }
gfCNCPoint5[2757] = {X 455.6724, Y 93.9777, Z -6.3333, A 0.000, B 0.000, C 0.000 }
gfCNCPoint5[2758] = {X 456.3743, Y 93.4663, Z -6.3333, A 0.000, B 0.000, C 0.000 }
gfCNCPoint5[2759] = {X 457.1672, Y 93.1118, Z -6.3333, A 0.000, B 0.000, C 0.000 }
gfCNCPoint5[2760] = {X 458.0163, Y 92.9296, Z -6.3333, A 0.000, B 0.000, C 0.000 }
gfCNCPoint5[2761] = {X 458.0163, Y 85.4858, Z -6.3333, A 0.000, B 0.000, C 0.000 }
gfCNCPoint5[2762] = {X 444.8418, Y 80.3214, Z -6.3333, A 0.000, B 0.000, C 0.000 }
gfCNCPoint5[2763] = {X 419.8634, Y 96.5017, Z -6.3333, A 0.000, B 0.000, C 0.000 }
gfCNCPoint5[2764] = {X 419.8667, Y 97.0654, Z -6.3333, A 0.000, B 0.000, C 0.000 }
gfCNCPoint5[2765] = {X 419.8667, Y 98.0000, Z -6.3333, A 0.000, B 0.000, C 0.000 }
gfCNCPoint5[2766] = {X 419.7624, Y 98.9257, Z -6.3333, A 0.000, B 0.000, C 0.000 }
gfCNCPoint5[2767] = {X 419.4547, Y 99.8050, Z -6.3333, A 0.000, B 0.000, C 0.000 }
gfCNCPoint5[2768] = {X 418.9591, Y 100.5937, Z -6.3333, A 0.000, B 0.000, C 0.000 }
gfCNCPoint5[2769] = {X 418.3004, Y 101.2524, Z -6.3333, A 0.000, B 0.000, C 0.000 }
gfCNCPoint5[2770] = {X 417.5117, Y 101.7480, Z -6.3333, A 0.000, B 0.000, C 0.000 }
gfCNCPoint5[2771] = {X 416.6324, Y 102.0557, Z -6.3333, A 0.000, B 0.000, C 0.000 }
gfCNCPoint5[2772] = {X 415.7067, Y 102.1600, Z -6.3333, A 0.000, B 0.000, C 0.000 }
gfCNCPoint5[2773] = {X 396.4059, Y 102.1600, Z -6.3333, A 0.000, B 0.000, C 0.000 }
gfCNCPoint5[2774] = {X 395.4803, Y 102.0557, Z -6.3333, A 0.000, B 0.000, C 0.000 }
gfCNCPoint5[2775] = {X 394.6010, Y 101.7480, Z -6.3333, A 0.000, B 0.000, C 0.000 }
gfCNCPoint5[2776] = {X 393.8122, Y 101.2524, Z -6.3333, A 0.000, B 0.000, C 0.000 }
gfCNCPoint5[2777] = {X 393.1535, Y 100.5937, Z -6.3333, A 0.000, B 0.000, C 0.000 }
gfCNCPoint5[2778] = {X 392.6579, Y 99.8050, Z -6.3333, A 0.000, B 0.000, C 0.000 }
gfCNCPoint5[2779] = {X 392.3502, Y 98.9257, Z -6.3333, A 0.000, B 0.000, C 0.000 }
gfCNCPoint5[2780] = {X 392.2459, Y 98.0000, Z -6.3333, A 0.000, B 0.000, C 0.000 }
gfCNCPoint5[2781] = {X 392.2459, Y 97.0659, Z -6.3333, A 0.000, B 0.000, C 0.000 }
gfCNCPoint5[2782] = {X 392.3504, Y 96.1396, Z -6.3333, A 0.000, B 0.000, C 0.000 }
gfCNCPoint5[2783] = {X 392.6585, Y 95.2597, Z -6.3333, A 0.000, B 0.000, C 0.000 }
gfCNCPoint5[2784] = {X 393.1548, Y 94.4706, Z -6.3333, A 0.000, B 0.000, C 0.000 }
gfCNCPoint5[2785] = {X 393.8144, Y 93.8118, Z -6.3333, A 0.000, B 0.000, C 0.000 }
gfCNCPoint5[2786] = {X 394.6042, Y 93.3164, Z -6.3333, A 0.000, B 0.000, C 0.000 }
gfCNCPoint5[2787] = {X 395.4844, Y 93.0093, Z -6.3333, A 0.000, B 0.000, C 0.000 }
gfCNCPoint5[2788] = {X 396.4109, Y 92.9059, Z -6.3333, A 0.000, B 0.000, C 0.000 }
gfCNCPoint5[2789] = {X 397.3636, Y 92.8626, Z -6.3333, A 0.000, B 0.000, C 0.000 }
gfCNCPoint5[2790] = {X 398.3131, Y 92.7724, Z -6.3333, A 0.000, B 0.000, C 0.000 }
gfCNCPoint5[2791] = {X 398.9990, Y 92.6061, Z -6.3333, A 0.000, B 0.000, C 0.000 }
gfCNCPoint5[2792] = {X 399.6307, Y 92.2912, Z -6.3333, A 0.000, B 0.000, C 0.000 }
gfCNCPoint5[2793] = {X 413.8851, Y 83.1630, Z -6.3333, A 0.000, B 0.000, C 0.000 }
gfCNCPoint5[2794] = {X 411.7280, Y 79.7945, Z -6.3333, A 0.000, B 0.000, C 0.000 }
gfCNCPoint5[2795] = {X 413.9282, Y 83.2304, Z -6.3333, A 0.000, B 0.000, C 0.000 }
gfCNCPoint5[2796] = {X 428.5794, Y 73.8480, Z -6.3333, A 0.000, B 0.000, C 0.000 }
gfCNCPoint5[2797] = {X 403.8433, Y 64.1432, Z -6.3333, A 0.000, B 0.000, C 0.000 }
gfCNCPoint5[2798] = {X 402.1208, Y 63.5730, Z -6.3333, A 0.000, B 0.000, C 0.000 }
gfCNCPoint5[2799] = {X 400.3461, Y 63.1951, Z -6.3333, A 0.000, B 0.000, C 0.000 }
gfCNCPoint5[2800] = {X 398.5408, Y 63.0140, Z -6.3333, A 0.000, B 0.000, C 0.000 }
gfCNCPoint5[2801] = {X 397.6404, Y 62.9096, Z -6.3333, A 0.000, B 0.000, C 0.000 }
gfCNCPoint5[2802] = {X 396.7853, Y 62.6090, Z -6.3333, A 0.000, B 0.000, C 0.000 }
gfCNCPoint5[2803] = {X 396.0177, Y 62.1269, Z -6.3333, A 0.000, B 0.000, C 0.000 }
gfCNCPoint5[2804] = {X 395.3754, Y 61.4873, Z -6.3333, A 0.000, B 0.000, C 0.000 }
gfCNCPoint5[2805] = {X 394.8902, Y 60.7217, Z -6.3333, A 0.000, B 0.000, C 0.000 }
gfCNCPoint5[2806] = {X 394.5860, Y 59.8679, Z -6.3333, A 0.000, B 0.000, C 0.000 }
gfCNCPoint5[2807] = {X 394.4779, Y 58.9680, Z -6.3333, A 0.000, B 0.000, C 0.000 }
gfCNCPoint5[2808] = {X 394.4777, Y 58.0000, Z -6.3333, A 0.000, B 0.000, C 0.000 }
gfCNCPoint5[2809] = {X 394.5800, Y 57.0921, Z -6.3333, A 0.000, B 0.000, C 0.000 }
gfCNCPoint5[2810] = {X 394.8818, Y 56.2298, Z -6.3333, A 0.000, B 0.000, C 0.000 }
gfCNCPoint5[2811] = {X 395.3678, Y 55.4562, Z -6.3333, A 0.000, B 0.000, C 0.000 }
gfCNCPoint5[2812] = {X 396.0139, Y 54.8101, Z -6.3333, A 0.000, B 0.000, C 0.000 }
gfCNCPoint5[2813] = {X 396.7875, Y 54.3240, Z -6.3333, A 0.000, B 0.000, C 0.000 }
gfCNCPoint5[2814] = {X 397.6498, Y 54.0223, Z -6.3333, A 0.000, B 0.000, C 0.000 }
gfCNCPoint5[2815] = {X 398.5577, Y 53.9200, Z -6.3333, A 0.000, B 0.000, C 0.000 }
gfCNCPoint5[2816] = {X 419.4886, Y 53.9200, Z -6.3333, A 0.000, B 0.000, C 0.000 }
gfCNCPoint5[2817] = {X 420.3965, Y 54.0223, Z -6.3333, A 0.000, B 0.000, C 0.000 }
gfCNCPoint5[2818] = {X 421.2589, Y 54.3240, Z -6.3333, A 0.000, B 0.000, C 0.000 }
gfCNCPoint5[2819] = {X 422.0324, Y 54.8101, Z -6.3333, A 0.000, B 0.000, C 0.000 }
gfCNCPoint5[2820] = {X 422.6785, Y 55.4562, Z -6.3333, A 0.000, B 0.000, C 0.000 }
gfCNCPoint5[2821] = {X 423.1646, Y 56.2298, Z -6.3333, A 0.000, B 0.000, C 0.000 }
gfCNCPoint5[2822] = {X 423.4663, Y 57.0921, Z -6.3333, A 0.000, B 0.000, C 0.000 }
gfCNCPoint5[2823] = {X 423.5686, Y 58.0000, Z -6.3333, A 0.000, B 0.000, C 0.000 }
gfCNCPoint5[2824] = {X 423.5686, Y 58.3958, Z -6.3333, A 0.000, B 0.000, C 0.000 }
gfCNCPoint5[2825] = {X 429.5238, Y 60.7161, Z -6.3333, A 0.000, B 0.000, C 0.000 }
gfCNCPoint5[2826] = {X 458.0981, Y 72.0535, Z -6.3333, A 0.000, B 0.000, C 0.000 }
gfCNCPoint5[2827] = {X 458.1004, Y 62.9982, Z -6.3333, A 0.000, B 0.000, C 0.000 }
gfCNCPoint5[2828] = {X 457.9640, Y 62.9839, Z -6.3333, A 0.000, B 0.000, C 0.000 }
gfCNCPoint5[2829] = {X 457.8281, Y 62.9649, Z -6.3333, A 0.000, B 0.000, C 0.000 }
gfCNCPoint5[2830] = {X 456.9087, Y 62.7078, Z -6.3333, A 0.000, B 0.000, C 0.000 }
gfCNCPoint5[2831] = {X 456.0742, Y 62.2441, Z -6.3333, A 0.000, B 0.000, C 0.000 }
gfCNCPoint5[2832] = {X 455.3703, Y 61.5992, Z -6.3333, A 0.000, B 0.000, C 0.000 }
gfCNCPoint5[2833] = {X 454.8356, Y 60.8084, Z -6.3333, A 0.000, B 0.000, C 0.000 }
gfCNCPoint5[2834] = {X 454.4993, Y 59.9149, Z -6.3333, A 0.000, B 0.000, C 0.000 }
gfCNCPoint5[2835] = {X 454.3797, Y 58.9678, Z -6.3333, A 0.000, B 0.000, C 0.000 }
gfCNCPoint5[2836] = {X 454.3796, Y 58.0000, Z -6.3333, A 0.000, B 0.000, C 0.000 }
gfCNCPoint5[2837] = {X 454.4819, Y 57.0921, Z -6.3333, A 0.000, B 0.000, C 0.000 }
gfCNCPoint5[2838] = {X 454.7837, Y 56.2298, Z -6.3333, A 0.000, B 0.000, C 0.000 }
gfCNCPoint5[2839] = {X 455.2697, Y 55.4562, Z -6.3333, A 0.000, B 0.000, C 0.000 }
gfCNCPoint5[2840] = {X 455.9158, Y 54.8101, Z -6.3333, A 0.000, B 0.000, C 0.000 }
gfCNCPoint5[2841] = {X 456.6894, Y 54.3240, Z -6.3333, A 0.000, B 0.000, C 0.000 }
gfCNCPoint5[2842] = {X 457.5517, Y 54.0223, Z -6.3333, A 0.000, B 0.000, C 0.000 }
gfCNCPoint5[2843] = {X 458.4596, Y 53.9200, Z -6.3333, A 0.000, B 0.000, C 0.000 }
gfCNCPoint5[2844] = {X 475.0000, Y 53.9200, Z -6.3333, A 0.000, B 0.000, C 0.000 }
gfCNCPoint5[2845] = {X 475.9079, Y 54.0223, Z -6.3333, A 0.000, B 0.000, C 0.000 }
gfCNCPoint5[2846] = {X 476.7702, Y 54.3240, Z -6.3333, A 0.000, B 0.000, C 0.000 }
gfCNCPoint5[2847] = {X 477.5438, Y 54.8101, Z -6.3333, A 0.000, B 0.000, C 0.000 }
gfCNCPoint5[2848] = {X 478.1899, Y 55.4562, Z -6.3333, A 0.000, B 0.000, C 0.000 }
gfCNCPoint5[2849] = {X 478.6760, Y 56.2298, Z -6.3333, A 0.000, B 0.000, C 0.000 }
gfCNCPoint5[2850] = {X 478.9777, Y 57.0921, Z -6.3333, A 0.000, B 0.000, C 0.000 }
gfCNCPoint5[2851] = {X 479.0800, Y 58.0000, Z -6.3333, A 0.000, B 0.000, C 0.000 }
gfCNCPoint5[2852] = {X 479.0800, Y 58.9342, Z -6.3333, A 0.000, B 0.000, C 0.000 }
gfCNCPoint5[2853] = {X 478.9888, Y 59.7917, Z -6.3333, A 0.000, B 0.000, C 0.000 }
gfCNCPoint5[2854] = {X 478.7195, Y 60.6109, Z -6.3333, A 0.000, B 0.000, C 0.000 }
gfCNCPoint5[2855] = {X 478.2840, Y 61.3551, Z -6.3333, A 0.000, B 0.000, C 0.000 }
gfCNCPoint5[2856] = {X 477.7018, Y 61.9913, Z -6.3333, A 0.000, B 0.000, C 0.000 }
gfCNCPoint5[2857] = {X 476.9990, Y 62.4908, Z -6.3333, A 0.000, B 0.000, C 0.000 }
gfCNCPoint5[2858] = {X 476.2068, Y 62.8315, Z -6.3333, A 0.000, B 0.000, C 0.000 }
gfCNCPoint5[2859] = {X 475.3607, Y 62.9981, Z -6.3333, A 0.000, B 0.000, C 0.000 }
gfCNCPoint5[2860] = {X 475.3612, Y 92.9626, Z -6.3333, A 0.000, B 0.000, C 0.000 }
gfCNCPoint5[2861] = {X 475.8364, Y 93.0717, Z -6.3333, A 0.000, B 0.000, C 0.000 }
gfCNCPoint5[2862] = {X 476.3038, Y 93.2109, Z -6.3333, A 0.000, B 0.000, C 0.000 }
gfCNCPoint5[2863] = {X 477.0721, Y 93.5592, Z -6.3333, A 0.000, B 0.000, C 0.000 }
gfCNCPoint5[2864] = {X 477.7518, Y 94.0588, Z -6.3333, A 0.000, B 0.000, C 0.000 }
gfCNCPoint5[2865] = {X 478.3136, Y 94.6881, Z -6.3333, A 0.000, B 0.000, C 0.000 }
gfCNCPoint5[2866] = {X 478.7331, Y 95.4199, Z -6.3333, A 0.000, B 0.000, C 0.000 }
gfCNCPoint5[2867] = {X 478.9923, Y 96.2227, Z -6.3333, A 0.000, B 0.000, C 0.000 }
gfCNCPoint5[2868] = {X 479.0800, Y 97.0617, Z -6.3333, A 0.000, B 0.000, C 0.000 }
gfCNCPoint5[2869] = {X 479.0800, Y 98.0000, Z -6.3333, A 0.000, B 0.000, C 0.000 }
gfCNCPoint5[2870] = {X 478.9777, Y 98.9079, Z -6.3333, A 0.000, B 0.000, C 0.000 }
gfCNCPoint5[2871] = {X 478.6760, Y 99.7702, Z -6.3333, A 0.000, B 0.000, C 0.000 }
gfCNCPoint5[2872] = {X 478.1899, Y 100.5438, Z -6.3333, A 0.000, B 0.000, C 0.000 }
gfCNCPoint5[2873] = {X 477.5438, Y 101.1899, Z -6.3333, A 0.000, B 0.000, C 0.000 }
gfCNCPoint5[2874] = {X 476.7702, Y 101.6760, Z -6.3333, A 0.000, B 0.000, C 0.000 }
gfCNCPoint5[2875] = {X 475.9079, Y 101.9777, Z -6.3333, A 0.000, B 0.000, C 0.000 }
gfCNCPoint5[2876] = {X 475.0000, Y 102.0800, Z -6.3333, A 0.000, B 0.000, C 0.000 }
gfCNCPoint5[2877] = {X 458.4596, Y 102.0800, Z -6.3333, A 0.000, B 0.000, C 0.000 }
gfCNCPoint5[2878] = {X 457.5517, Y 101.9777, Z -6.3333, A 0.000, B 0.000, C 0.000 }
gfCNCPoint5[2879] = {X 456.6894, Y 101.6760, Z -6.3333, A 0.000, B 0.000, C 0.000 }
gfCNCPoint5[2880] = {X 455.9158, Y 101.1899, Z -6.3333, A 0.000, B 0.000, C 0.000 }
gfCNCPoint5[2881] = {X 455.2697, Y 100.5438, Z -6.3333, A 0.000, B 0.000, C 0.000 }
gfCNCPoint5[2882] = {X 454.7837, Y 99.7702, Z -6.3333, A 0.000, B 0.000, C 0.000 }
gfCNCPoint5[2883] = {X 454.4819, Y 98.9079, Z -6.3333, A 0.000, B 0.000, C 0.000 }
gfCNCPoint5[2884] = {X 454.3796, Y 98.0000, Z -6.3333, A 0.000, B 0.000, C 0.000 }
gfCNCPoint5[2885] = {X 454.3796, Y 97.0659, Z -6.3333, A 0.000, B 0.000, C 0.000 }
gfCNCPoint5[2886] = {X 454.4707, Y 96.2088, Z -6.3333, A 0.000, B 0.000, C 0.000 }
gfCNCPoint5[2887] = {X 454.7398, Y 95.3899, Z -6.3333, A 0.000, B 0.000, C 0.000 }
gfCNCPoint5[2888] = {X 455.1749, Y 94.6458, Z -6.3333, A 0.000, B 0.000, C 0.000 }
gfCNCPoint5[2889] = {X 455.7566, Y 94.0098, Z -6.3333, A 0.000, B 0.000, C 0.000 }
gfCNCPoint5[2890] = {X 456.4590, Y 93.5101, Z -6.3333, A 0.000, B 0.000, C 0.000 }
gfCNCPoint5[2891] = {X 457.2507, Y 93.1692, Z -6.3333, A 0.000, B 0.000, C 0.000 }
gfCNCPoint5[2892] = {X 458.0963, Y 93.0021, Z -6.3333, A 0.000, B 0.000, C 0.000 }
gfCNCPoint5[2893] = {X 458.0963, Y 85.4313, Z -6.3333, A 0.000, B 0.000, C 0.000 }
gfCNCPoint5[2894] = {X 444.8327, Y 80.2319, Z -6.3333, A 0.000, B 0.000, C 0.000 }
gfCNCPoint5[2895] = {X 419.7832, Y 96.4584, Z -6.3333, A 0.000, B 0.000, C 0.000 }
gfCNCPoint5[2896] = {X 419.7867, Y 97.0657, Z -6.3333, A 0.000, B 0.000, C 0.000 }
gfCNCPoint5[2897] = {X 419.7867, Y 98.0000, Z -6.3333, A 0.000, B 0.000, C 0.000 }
gfCNCPoint5[2898] = {X 419.6844, Y 98.9079, Z -6.3333, A 0.000, B 0.000, C 0.000 }
gfCNCPoint5[2899] = {X 419.3827, Y 99.7702, Z -6.3333, A 0.000, B 0.000, C 0.000 }
gfCNCPoint5[2900] = {X 418.8966, Y 100.5438, Z -6.3333, A 0.000, B 0.000, C 0.000 }
gfCNCPoint5[2901] = {X 418.2505, Y 101.1899, Z -6.3333, A 0.000, B 0.000, C 0.000 }
gfCNCPoint5[2902] = {X 417.4769, Y 101.6760, Z -6.3333, A 0.000, B 0.000, C 0.000 }
gfCNCPoint5[2903] = {X 416.6146, Y 101.9777, Z -6.3333, A 0.000, B 0.000, C 0.000 }
gfCNCPoint5[2904] = {X 415.7067, Y 102.0800, Z -6.3333, A 0.000, B 0.000, C 0.000 }
gfCNCPoint5[2905] = {X 396.4059, Y 102.0800, Z -6.3333, A 0.000, B 0.000, C 0.000 }
gfCNCPoint5[2906] = {X 395.4981, Y 101.9777, Z -6.3333, A 0.000, B 0.000, C 0.000 }
gfCNCPoint5[2907] = {X 394.6357, Y 101.6760, Z -6.3333, A 0.000, B 0.000, C 0.000 }
gfCNCPoint5[2908] = {X 393.8621, Y 101.1899, Z -6.3333, A 0.000, B 0.000, C 0.000 }
gfCNCPoint5[2909] = {X 393.2161, Y 100.5438, Z -6.3333, A 0.000, B 0.000, C 0.000 }
gfCNCPoint5[2910] = {X 392.7300, Y 99.7702, Z -6.3333, A 0.000, B 0.000, C 0.000 }
gfCNCPoint5[2911] = {X 392.4282, Y 98.9079, Z -6.3333, A 0.000, B 0.000, C 0.000 }
gfCNCPoint5[2912] = {X 392.3259, Y 98.0000, Z -6.3333, A 0.000, B 0.000, C 0.000 }
gfCNCPoint5[2913] = {X 392.3259, Y 97.0659, Z -6.3333, A 0.000, B 0.000, C 0.000 }
gfCNCPoint5[2914] = {X 392.4284, Y 96.1573, Z -6.3333, A 0.000, B 0.000, C 0.000 }
gfCNCPoint5[2915] = {X 392.7307, Y 95.2942, Z -6.3333, A 0.000, B 0.000, C 0.000 }
gfCNCPoint5[2916] = {X 393.2176, Y 94.5202, Z -6.3333, A 0.000, B 0.000, C 0.000 }
gfCNCPoint5[2917] = {X 393.8647, Y 93.8740, Z -6.3333, A 0.000, B 0.000, C 0.000 }
gfCNCPoint5[2918] = {X 394.6394, Y 93.3882, Z -6.3333, A 0.000, B 0.000, C 0.000 }
gfCNCPoint5[2919] = {X 395.5028, Y 93.0871, Z -6.3333, A 0.000, B 0.000, C 0.000 }
gfCNCPoint5[2920] = {X 396.4117, Y 92.9859, Z -6.3333, A 0.000, B 0.000, C 0.000 }
gfCNCPoint5[2921] = {X 397.3689, Y 92.9424, Z -6.3333, A 0.000, B 0.000, C 0.000 }
gfCNCPoint5[2922] = {X 398.3229, Y 92.8518, Z -6.3333, A 0.000, B 0.000, C 0.000 }
gfCNCPoint5[2923] = {X 399.0264, Y 92.6813, Z -6.3333, A 0.000, B 0.000, C 0.000 }
gfCNCPoint5[2924] = {X 399.6742, Y 92.3584, Z -6.3333, A 0.000, B 0.000, C 0.000 }
gfCNCPoint5[2925] = {X 413.9282, Y 83.2304, Z -6.3333, A 0.000, B 0.000, C 0.000 }
gfCNCPoint5[2926] = {X 411.7650, Y 79.8523, Z -6.3333, A 0.000, B 0.000, C 0.000 }
gfCNCPoint5[2927] = {X 411.7672, Y 79.8509, Z -6.3333, A 0.000, B 0.000, C 0.000 }
gfCNCPoint5[2928] = {X 413.9652, Y 83.2882, Z -6.3333, A 0.000, B 0.000, C 0.000 }
gfCNCPoint5[2929] = {X 428.7548, Y 73.8308, Z -6.3333, A 0.000, B 0.000, C 0.000 }
gfCNCPoint5[2930] = {X 403.8726, Y 64.0687, Z -6.3333, A 0.000, B 0.000, C 0.000 }
gfCNCPoint5[2931] = {X 402.1412, Y 63.4957, Z -6.3333, A 0.000, B 0.000, C 0.000 }
gfCNCPoint5[2932] = {X 400.3574, Y 63.1159, Z -6.3333, A 0.000, B 0.000, C 0.000 }
gfCNCPoint5[2933] = {X 398.5427, Y 62.9340, Z -6.3333, A 0.000, B 0.000, C 0.000 }
gfCNCPoint5[2934] = {X 397.6551, Y 62.8309, Z -6.3333, A 0.000, B 0.000, C 0.000 }
gfCNCPoint5[2935] = {X 396.8125, Y 62.5333, Z -6.3333, A 0.000, B 0.000, C 0.000 }
gfCNCPoint5[2936] = {X 396.0571, Y 62.0560, Z -6.3333, A 0.000, B 0.000, C 0.000 }
gfCNCPoint5[2937] = {X 395.4264, Y 61.4230, Z -6.3333, A 0.000, B 0.000, C 0.000 }
gfCNCPoint5[2938] = {X 394.9520, Y 60.6657, Z -6.3333, A 0.000, B 0.000, C 0.000 }
gfCNCPoint5[2939] = {X 394.6575, Y 59.8221, Z -6.3333, A 0.000, B 0.000, C 0.000 }
gfCNCPoint5[2940] = {X 394.5577, Y 58.9341, Z -6.3333, A 0.000, B 0.000, C 0.000 }
gfCNCPoint5[2941] = {X 394.5577, Y 58.0000, Z -6.3333, A 0.000, B 0.000, C 0.000 }
gfCNCPoint5[2942] = {X 394.6580, Y 57.1099, Z -6.3333, A 0.000, B 0.000, C 0.000 }
gfCNCPoint5[2943] = {X 394.9538, Y 56.2645, Z -6.3333, A 0.000, B 0.000, C 0.000 }
gfCNCPoint5[2944] = {X 395.4304, Y 55.5060, Z -6.3333, A 0.000, B 0.000, C 0.000 }
gfCNCPoint5[2945] = {X 396.0638, Y 54.8727, Z -6.3333, A 0.000, B 0.000, C 0.000 }
gfCNCPoint5[2946] = {X 396.8222, Y 54.3961, Z -6.3333, A 0.000, B 0.000, C 0.000 }
gfCNCPoint5[2947] = {X 397.6676, Y 54.1003, Z -6.3333, A 0.000, B 0.000, C 0.000 }
gfCNCPoint5[2948] = {X 398.5577, Y 54.0000, Z -6.3333, A 0.000, B 0.000, C 0.000 }
gfCNCPoint5[2949] = {X 419.4886, Y 54.0000, Z -6.3333, A 0.000, B 0.000, C 0.000 }
gfCNCPoint5[2950] = {X 420.3787, Y 54.1003, Z -6.3333, A 0.000, B 0.000, C 0.000 }
gfCNCPoint5[2951] = {X 421.2241, Y 54.3961, Z -6.3333, A 0.000, B 0.000, C 0.000 }
gfCNCPoint5[2952] = {X 421.9826, Y 54.8727, Z -6.3333, A 0.000, B 0.000, C 0.000 }
gfCNCPoint5[2953] = {X 422.6159, Y 55.5060, Z -6.3333, A 0.000, B 0.000, C 0.000 }
gfCNCPoint5[2954] = {X 423.0925, Y 56.2645, Z -6.3333, A 0.000, B 0.000, C 0.000 }
gfCNCPoint5[2955] = {X 423.3883, Y 57.1099, Z -6.3333, A 0.000, B 0.000, C 0.000 }
gfCNCPoint5[2956] = {X 423.4886, Y 58.0000, Z -6.3333, A 0.000, B 0.000, C 0.000 }
gfCNCPoint5[2957] = {X 423.4886, Y 58.4505, Z -6.3333, A 0.000, B 0.000, C 0.000 }
gfCNCPoint5[2958] = {X 429.4945, Y 60.7905, Z -6.3333, A 0.000, B 0.000, C 0.000 }
gfCNCPoint5[2959] = {X 458.1781, Y 72.1713, Z -6.3333, A 0.000, B 0.000, C 0.000 }
gfCNCPoint5[2960] = {X 458.1786, Y 63.0391, Z -6.3333, A 0.000, B 0.000, C 0.000 }
gfCNCPoint5[2961] = {X 458.1841, Y 62.9246, Z -6.3333, A 0.000, B 0.000, C 0.000 }
gfCNCPoint5[2962] = {X 458.0118, Y 62.9089, Z -6.3333, A 0.000, B 0.000, C 0.000 }
gfCNCPoint5[2963] = {X 457.8405, Y 62.8859, Z -6.3333, A 0.000, B 0.000, C 0.000 }
gfCNCPoint5[2964] = {X 456.9340, Y 62.6317, Z -6.3333, A 0.000, B 0.000, C 0.000 }
gfCNCPoint5[2965] = {X 456.1121, Y 62.1727, Z -6.3333, A 0.000, B 0.000, C 0.000 }
gfCNCPoint5[2966] = {X 455.4201, Y 61.5344, Z -6.3333, A 0.000, B 0.000, C 0.000 }
gfCNCPoint5[2967] = {X 454.8966, Y 60.7520, Z -6.3333, A 0.000, B 0.000, C 0.000 }
gfCNCPoint5[2968] = {X 454.5704, Y 59.8689, Z -6.3333, A 0.000, B 0.000, C 0.000 }
gfCNCPoint5[2969] = {X 454.4596, Y 58.9341, Z -6.3333, A 0.000, B 0.000, C 0.000 }
gfCNCPoint5[2970] = {X 454.4596, Y 58.0000, Z -6.3333, A 0.000, B 0.000, C 0.000 }
gfCNCPoint5[2971] = {X 454.5599, Y 57.1099, Z -6.3333, A 0.000, B 0.000, C 0.000 }
gfCNCPoint5[2972] = {X 454.8557, Y 56.2645, Z -6.3333, A 0.000, B 0.000, C 0.000 }
gfCNCPoint5[2973] = {X 455.3323, Y 55.5060, Z -6.3333, A 0.000, B 0.000, C 0.000 }
gfCNCPoint5[2974] = {X 455.9656, Y 54.8727, Z -6.3333, A 0.000, B 0.000, C 0.000 }
gfCNCPoint5[2975] = {X 456.7241, Y 54.3961, Z -6.3333, A 0.000, B 0.000, C 0.000 }
gfCNCPoint5[2976] = {X 457.5695, Y 54.1003, Z -6.3333, A 0.000, B 0.000, C 0.000 }
gfCNCPoint5[2977] = {X 458.4596, Y 54.0000, Z -6.3333, A 0.000, B 0.000, C 0.000 }
gfCNCPoint5[2978] = {X 475.0000, Y 54.0000, Z -6.3333, A 0.000, B 0.000, C 0.000 }
gfCNCPoint5[2979] = {X 475.8901, Y 54.1003, Z -6.3333, A 0.000, B 0.000, C 0.000 }
gfCNCPoint5[2980] = {X 476.7355, Y 54.3961, Z -6.3333, A 0.000, B 0.000, C 0.000 }
gfCNCPoint5[2981] = {X 477.4940, Y 54.8727, Z -6.3333, A 0.000, B 0.000, C 0.000 }
gfCNCPoint5[2982] = {X 478.1273, Y 55.5060, Z -6.3333, A 0.000, B 0.000, C 0.000 }
gfCNCPoint5[2983] = {X 478.6039, Y 56.2645, Z -6.3333, A 0.000, B 0.000, C 0.000 }
gfCNCPoint5[2984] = {X 478.8997, Y 57.1099, Z -6.3333, A 0.000, B 0.000, C 0.000 }
gfCNCPoint5[2985] = {X 479.0000, Y 58.0000, Z -6.3333, A 0.000, B 0.000, C 0.000 }
gfCNCPoint5[2986] = {X 478.9999, Y 58.9671, Z -6.3333, A 0.000, B 0.000, C 0.000 }
gfCNCPoint5[2987] = {X 478.9023, Y 59.8126, Z -6.3333, A 0.000, B 0.000, C 0.000 }
gfCNCPoint5[2988] = {X 478.6281, Y 60.6184, Z -6.3333, A 0.000, B 0.000, C 0.000 }
gfCNCPoint5[2989] = {X 478.1896, Y 61.3478, Z -6.3333, A 0.000, B 0.000, C 0.000 }
gfCNCPoint5[2990] = {X 477.6067, Y 61.9680, Z -6.3333, A 0.000, B 0.000, C 0.000 }
gfCNCPoint5[2991] = {X 476.9058, Y 62.4509, Z -6.3333, A 0.000, B 0.000, C 0.000 }
gfCNCPoint5[2992] = {X 476.1186, Y 62.7745, Z -6.3333, A 0.000, B 0.000, C 0.000 }
gfCNCPoint5[2993] = {X 475.2807, Y 62.9242, Z -6.3333, A 0.000, B 0.000, C 0.000 }
gfCNCPoint5[2994] = {X 475.2812, Y 93.0287, Z -6.3333, A 0.000, B 0.000, C 0.000 }
gfCNCPoint5[2995] = {X 475.7842, Y 93.1408, Z -6.3333, A 0.000, B 0.000, C 0.000 }
gfCNCPoint5[2996] = {X 476.2785, Y 93.2868, Z -6.3333, A 0.000, B 0.000, C 0.000 }
gfCNCPoint5[2997] = {X 477.0316, Y 93.6283, Z -6.3333, A 0.000, B 0.000, C 0.000 }
gfCNCPoint5[2998] = {X 477.6980, Y 94.1180, Z -6.3333, A 0.000, B 0.000, C 0.000 }
gfCNCPoint5[2999] = {X 478.2487, Y 94.7349, Z -6.3333, A 0.000, B 0.000, C 0.000 }
gfCNCPoint5[3000] = {X 478.6600, Y 95.4523, Z -6.3333, A 0.000, B 0.000, C 0.000 }
gfCNCPoint5[3001] = {X 478.9141, Y 96.2392, Z -6.3333, A 0.000, B 0.000, C 0.000 }
gfCNCPoint5[3002] = {X 479.0000, Y 97.0617, Z -6.3333, A 0.000, B 0.000, C 0.000 }
gfCNCPoint5[3003] = {X 479.0000, Y 98.0000, Z -6.3333, A 0.000, B 0.000, C 0.000 }
gfCNCPoint5[3004] = {X 478.8997, Y 98.8901, Z -6.3333, A 0.000, B 0.000, C 0.000 }
gfCNCPoint5[3005] = {X 478.6039, Y 99.7355, Z -6.3333, A 0.000, B 0.000, C 0.000 }
gfCNCPoint5[3006] = {X 478.1273, Y 100.4940, Z -6.3333, A 0.000, B 0.000, C 0.000 }
gfCNCPoint5[3007] = {X 477.4940, Y 101.1273, Z -6.3333, A 0.000, B 0.000, C 0.000 }
gfCNCPoint5[3008] = {X 476.7355, Y 101.6039, Z -6.3333, A 0.000, B 0.000, C 0.000 }
gfCNCPoint5[3009] = {X 475.8901, Y 101.8997, Z -6.3333, A 0.000, B 0.000, C 0.000 }
gfCNCPoint5[3010] = {X 475.0000, Y 102.0000, Z -6.3333, A 0.000, B 0.000, C 0.000 }
gfCNCPoint5[3011] = {X 458.4596, Y 102.0000, Z -6.3333, A 0.000, B 0.000, C 0.000 }
gfCNCPoint5[3012] = {X 457.5695, Y 101.8997, Z -6.3333, A 0.000, B 0.000, C 0.000 }
gfCNCPoint5[3013] = {X 456.7241, Y 101.6039, Z -6.3333, A 0.000, B 0.000, C 0.000 }
gfCNCPoint5[3014] = {X 455.9656, Y 101.1273, Z -6.3333, A 0.000, B 0.000, C 0.000 }
gfCNCPoint5[3015] = {X 455.3323, Y 100.4940, Z -6.3333, A 0.000, B 0.000, C 0.000 }
gfCNCPoint5[3016] = {X 454.8557, Y 99.7355, Z -6.3333, A 0.000, B 0.000, C 0.000 }
gfCNCPoint5[3017] = {X 454.5599, Y 98.8901, Z -6.3333, A 0.000, B 0.000, C 0.000 }
gfCNCPoint5[3018] = {X 454.4596, Y 98.0000, Z -6.3333, A 0.000, B 0.000, C 0.000 }
gfCNCPoint5[3019] = {X 454.4596, Y 97.0659, Z -6.3333, A 0.000, B 0.000, C 0.000 }
gfCNCPoint5[3020] = {X 454.5511, Y 96.2154, Z -6.3333, A 0.000, B 0.000, C 0.000 }
gfCNCPoint5[3021] = {X 454.8213, Y 95.4037, Z -6.3333, A 0.000, B 0.000, C 0.000 }
gfCNCPoint5[3022] = {X 455.2580, Y 94.6681, Z -6.3333, A 0.000, B 0.000, C 0.000 }
gfCNCPoint5[3023] = {X 455.8411, Y 94.0422, Z -6.3333, A 0.000, B 0.000, C 0.000 }
gfCNCPoint5[3024] = {X 456.5439, Y 93.5545, Z -6.3333, A 0.000, B 0.000, C 0.000 }
gfCNCPoint5[3025] = {X 457.3344, Y 93.2275, Z -6.3333, A 0.000, B 0.000, C 0.000 }
gfCNCPoint5[3026] = {X 458.1763, Y 93.0760, Z -6.3333, A 0.000, B 0.000, C 0.000 }
gfCNCPoint5[3027] = {X 458.1763, Y 85.3767, Z -6.3333, A 0.000, B 0.000, C 0.000 }
gfCNCPoint5[3028] = {X 445.0148, Y 80.2174, Z -6.3333, A 0.000, B 0.000, C 0.000 }
gfCNCPoint5[3029] = {X 444.8242, Y 80.1421, Z -6.3333, A 0.000, B 0.000, C 0.000 }
gfCNCPoint5[3030] = {X 419.7029, Y 96.4151, Z -6.3333, A 0.000, B 0.000, C 0.000 }
gfCNCPoint5[3031] = {X 419.7067, Y 97.0659, Z -6.3333, A 0.000, B 0.000, C 0.000 }
gfCNCPoint5[3032] = {X 419.7067, Y 98.0000, Z -6.3333, A 0.000, B 0.000, C 0.000 }
gfCNCPoint5[3033] = {X 419.6064, Y 98.8901, Z -6.3333, A 0.000, B 0.000, C 0.000 }
gfCNCPoint5[3034] = {X 419.3106, Y 99.7355, Z -6.3333, A 0.000, B 0.000, C 0.000 }
gfCNCPoint5[3035] = {X 418.8340, Y 100.4940, Z -6.3333, A 0.000, B 0.000, C 0.000 }
gfCNCPoint5[3036] = {X 418.2007, Y 101.1273, Z -6.3333, A 0.000, B 0.000, C 0.000 }
gfCNCPoint5[3037] = {X 417.4422, Y 101.6039, Z -6.3333, A 0.000, B 0.000, C 0.000 }
gfCNCPoint5[3038] = {X 416.5968, Y 101.8997, Z -6.3333, A 0.000, B 0.000, C 0.000 }
gfCNCPoint5[3039] = {X 415.7067, Y 102.0000, Z -6.3333, A 0.000, B 0.000, C 0.000 }
gfCNCPoint5[3040] = {X 396.4059, Y 102.0000, Z -6.3333, A 0.000, B 0.000, C 0.000 }
gfCNCPoint5[3041] = {X 395.5159, Y 101.8997, Z -6.3333, A 0.000, B 0.000, C 0.000 }
gfCNCPoint5[3042] = {X 394.6704, Y 101.6039, Z -6.3333, A 0.000, B 0.000, C 0.000 }
gfCNCPoint5[3043] = {X 393.9120, Y 101.1273, Z -6.3333, A 0.000, B 0.000, C 0.000 }
gfCNCPoint5[3044] = {X 393.2786, Y 100.4940, Z -6.3333, A 0.000, B 0.000, C 0.000 }
gfCNCPoint5[3045] = {X 392.8021, Y 99.7355, Z -6.3333, A 0.000, B 0.000, C 0.000 }
gfCNCPoint5[3046] = {X 392.5062, Y 98.8901, Z -6.3333, A 0.000, B 0.000, C 0.000 }
gfCNCPoint5[3047] = {X 392.4059, Y 98.0000, Z -6.3333, A 0.000, B 0.000, C 0.000 }
gfCNCPoint5[3048] = {X 392.4059, Y 97.0659, Z -6.3333, A 0.000, B 0.000, C 0.000 }
gfCNCPoint5[3049] = {X 392.5064, Y 96.1749, Z -6.3333, A 0.000, B 0.000, C 0.000 }
gfCNCPoint5[3050] = {X 392.8029, Y 95.3287, Z -6.3333, A 0.000, B 0.000, C 0.000 }
gfCNCPoint5[3051] = {X 393.2804, Y 94.5698, Z -6.3333, A 0.000, B 0.000, C 0.000 }
gfCNCPoint5[3052] = {X 393.9149, Y 93.9363, Z -6.3333, A 0.000, B 0.000, C 0.000 }
gfCNCPoint5[3053] = {X 394.6746, Y 93.4600, Z -6.3333, A 0.000, B 0.000, C 0.000 }
gfCNCPoint5[3054] = {X 395.5213, Y 93.1650, Z -6.3333, A 0.000, B 0.000, C 0.000 }
gfCNCPoint5[3055] = {X 396.4125, Y 93.0659, Z -6.3333, A 0.000, B 0.000, C 0.000 }
gfCNCPoint5[3056] = {X 397.3742, Y 93.0222, Z -6.3333, A 0.000, B 0.000, C 0.000 }
gfCNCPoint5[3057] = {X 398.3327, Y 92.9312, Z -6.3333, A 0.000, B 0.000, C 0.000 }
gfCNCPoint5[3058] = {X 399.0537, Y 92.7564, Z -6.3333, A 0.000, B 0.000, C 0.000 }
gfCNCPoint5[3059] = {X 399.7177, Y 92.4255, Z -6.3333, A 0.000, B 0.000, C 0.000 }
gfCNCPoint5[3060] = {X 405.2576, Y 88.8564, Z -6.3333, A 0.000, B 0.000, C 0.000 }
gfCNCPoint5[3061] = {X 413.9652, Y 83.2882, Z -6.3333, A 0.000, B 0.000, C 0.000 }
gfCNCPoint5[3062] = {X 411.7672, Y 79.8509, Z -6.3333, A 0.000, B 0.000, C 0.000 }
gfCNCPoint5[3063] = {X 411.7672, Y 79.8509, Z -3.3333, A 0.000, B 0.000, C 0.000 }
gfCNCPoint5[3064] = {X 411.7672, Y 79.8509, Z 11.0000, A 0.000, B 0.000, C 0.000 }
gfCNCPoint5[3065] = {X 466.3114, Y 28.5934, Z 11.0000, A 0.000, B 0.000, C 0.000 }
gfCNCPoint5[3066] = {X 466.3114, Y 28.5934, Z -3.3333, A 0.000, B 0.000, C 0.000 }
gfCNCPoint5[3067] = {X 466.3114, Y 28.5934, Z -6.3333, A 0.000, B 0.000, C 0.000 }
gfCNCPoint5[3068] = {X 462.2314, Y 28.5935, Z -6.3333, A 0.000, B 0.000, C 0.000 }
gfCNCPoint5[3069] = {X 462.2317, Y 40.9139, Z -6.3333, A 0.000, B 0.000, C 0.000 }
gfCNCPoint5[3070] = {X 462.2401, Y 40.9209, Z -6.3333, A 0.000, B 0.000, C 0.000 }
gfCNCPoint5[3071] = {X 462.8747, Y 41.5913, Z -6.3333, A 0.000, B 0.000, C 0.000 }
gfCNCPoint5[3072] = {X 463.3524, Y 42.3813, Z -6.3333, A 0.000, B 0.000, C 0.000 }
gfCNCPoint5[3073] = {X 463.6513, Y 43.2548, Z -6.3333, A 0.000, B 0.000, C 0.000 }
gfCNCPoint5[3074] = {X 463.7578, Y 44.1718, Z -6.3333, A 0.000, B 0.000, C 0.000 }
gfCNCPoint5[3075] = {X 463.7579, Y 45.0000, Z -6.3333, A 0.000, B 0.000, C 0.000 }
gfCNCPoint5[3076] = {X 463.6496, Y 45.9613, Z -6.3333, A 0.000, B 0.000, C 0.000 }
gfCNCPoint5[3077] = {X 463.3301, Y 46.8744, Z -6.3333, A 0.000, B 0.000, C 0.000 }
gfCNCPoint5[3078] = {X 462.8155, Y 47.6935, Z -6.3333, A 0.000, B 0.000, C 0.000 }
gfCNCPoint5[3079] = {X 462.1314, Y 48.3775, Z -6.3333, A 0.000, B 0.000, C 0.000 }
gfCNCPoint5[3080] = {X 461.3123, Y 48.8922, Z -6.3333, A 0.000, B 0.000, C 0.000 }
gfCNCPoint5[3081] = {X 460.3992, Y 49.2117, Z -6.3333, A 0.000, B 0.000, C 0.000 }
gfCNCPoint5[3082] = {X 459.4379, Y 49.3200, Z -6.3333, A 0.000, B 0.000, C 0.000 }
gfCNCPoint5[3083] = {X 452.9945, Y 49.3200, Z -6.3333, A 0.000, B 0.000, C 0.000 }
gfCNCPoint5[3084] = {X 452.0380, Y 49.2128, Z -6.3333, A 0.000, B 0.000, C 0.000 }
gfCNCPoint5[3085] = {X 451.1291, Y 48.8965, Z -6.3333, A 0.000, B 0.000, C 0.000 }
gfCNCPoint5[3086] = {X 450.3127, Y 48.3868, Z -6.3333, A 0.000, B 0.000, C 0.000 }
gfCNCPoint5[3087] = {X 449.6294, Y 47.7091, Z -6.3333, A 0.000, B 0.000, C 0.000 }
gfCNCPoint5[3088] = {X 449.1132, Y 46.8968, Z -6.3333, A 0.000, B 0.000, C 0.000 }
gfCNCPoint5[3089] = {X 448.7895, Y 45.9905, Z -6.3333, A 0.000, B 0.000, C 0.000 }
gfCNCPoint5[3090] = {X 448.6746, Y 45.0349, Z -6.3333, A 0.000, B 0.000, C 0.000 }
gfCNCPoint5[3091] = {X 448.6749, Y 44.1494, Z -6.3333, A 0.000, B 0.000, C 0.000 }
gfCNCPoint5[3092] = {X 448.7853, Y 43.2364, Z -6.3333, A 0.000, B 0.000, C 0.000 }
gfCNCPoint5[3093] = {X 449.0865, Y 42.3675, Z -6.3333, A 0.000, B 0.000, C 0.000 }
gfCNCPoint5[3094] = {X 449.5648, Y 41.5821, Z -6.3333, A 0.000, B 0.000, C 0.000 }
gfCNCPoint5[3095] = {X 450.1984, Y 40.9157, Z -6.3333, A 0.000, B 0.000, C 0.000 }
gfCNCPoint5[3096] = {X 450.1984, Y 34.4738, Z -6.3333, A 0.000, B 0.000, C 0.000 }
gfCNCPoint5[3097] = {X 447.4753, Y 34.4738, Z -6.3333, A 0.000, B 0.000, C 0.000 }
gfCNCPoint5[3098] = {X 443.1900, Y 42.8174, Z -6.3333, A 0.000, B 0.000, C 0.000 }
gfCNCPoint5[3099] = {X 443.1948, Y 42.8309, Z -6.3333, A 0.000, B 0.000, C 0.000 }
gfCNCPoint5[3100] = {X 443.3605, Y 43.4917, Z -6.3333, A 0.000, B 0.000, C 0.000 }
gfCNCPoint5[3101] = {X 443.4203, Y 44.1703, Z -6.3333, A 0.000, B 0.000, C 0.000 }
gfCNCPoint5[3102] = {X 443.4205, Y 45.0000, Z -6.3333, A 0.000, B 0.000, C 0.000 }
gfCNCPoint5[3103] = {X 443.3122, Y 45.9613, Z -6.3333, A 0.000, B 0.000, C 0.000 }
gfCNCPoint5[3104] = {X 442.9927, Y 46.8744, Z -6.3333, A 0.000, B 0.000, C 0.000 }
gfCNCPoint5[3105] = {X 442.4780, Y 47.6935, Z -6.3333, A 0.000, B 0.000, C 0.000 }
gfCNCPoint5[3106] = {X 441.7939, Y 48.3775, Z -6.3333, A 0.000, B 0.000, C 0.000 }
gfCNCPoint5[3107] = {X 440.9748, Y 48.8922, Z -6.3333, A 0.000, B 0.000, C 0.000 }
gfCNCPoint5[3108] = {X 440.0618, Y 49.2117, Z -6.3333, A 0.000, B 0.000, C 0.000 }
gfCNCPoint5[3109] = {X 439.1005, Y 49.3200, Z -6.3333, A 0.000, B 0.000, C 0.000 }
gfCNCPoint5[3110] = {X 432.5144, Y 49.3200, Z -6.3333, A 0.000, B 0.000, C 0.000 }
gfCNCPoint5[3111] = {X 431.5531, Y 49.2117, Z -6.3333, A 0.000, B 0.000, C 0.000 }
gfCNCPoint5[3112] = {X 430.6401, Y 48.8922, Z -6.3333, A 0.000, B 0.000, C 0.000 }
gfCNCPoint5[3113] = {X 429.8210, Y 48.3775, Z -6.3333, A 0.000, B 0.000, C 0.000 }
gfCNCPoint5[3114] = {X 429.1369, Y 47.6935, Z -6.3333, A 0.000, B 0.000, C 0.000 }
gfCNCPoint5[3115] = {X 428.6223, Y 46.8745, Z -6.3333, A 0.000, B 0.000, C 0.000 }
gfCNCPoint5[3116] = {X 428.3027, Y 45.9614, Z -6.3333, A 0.000, B 0.000, C 0.000 }
gfCNCPoint5[3117] = {X 428.1944, Y 45.0001, Z -6.3333, A 0.000, B 0.000, C 0.000 }
gfCNCPoint5[3118] = {X 428.1948, Y 44.1494, Z -6.3333, A 0.000, B 0.000, C 0.000 }
gfCNCPoint5[3119] = {X 428.2925, Y 43.2935, Z -6.3333, A 0.000, B 0.000, C 0.000 }
gfCNCPoint5[3120] = {X 428.5580, Y 42.4740, Z -6.3333, A 0.000, B 0.000, C 0.000 }
gfCNCPoint5[3121] = {X 428.9809, Y 41.7236, Z -6.3333, A 0.000, B 0.000, C 0.000 }
gfCNCPoint5[3122] = {X 429.5442, Y 41.0719, Z -6.3333, A 0.000, B 0.000, C 0.000 }
gfCNCPoint5[3123] = {X 430.2256, Y 40.5449, Z -6.3333, A 0.000, B 0.000, C 0.000 }
gfCNCPoint5[3124] = {X 430.9981, Y 40.1637, Z -6.3333, A 0.000, B 0.000, C 0.000 }
gfCNCPoint5[3125] = {X 434.9868, Y 32.3561, Z -6.3333, A 0.000, B 0.000, C 0.000 }
gfCNCPoint5[3126] = {X 433.8227, Y 31.5745, Z -6.3333, A 0.000, B 0.000, C 0.000 }
gfCNCPoint5[3127] = {X 432.7641, Y 30.6549, Z -6.3333, A 0.000, B 0.000, C 0.000 }
gfCNCPoint5[3128] = {X 431.8274, Y 29.6116, Z -6.3333, A 0.000, B 0.000, C 0.000 }
gfCNCPoint5[3129] = {X 431.0268, Y 28.4604, Z -6.3333, A 0.000, B 0.000, C 0.000 }
gfCNCPoint5[3130] = {X 430.3747, Y 27.2190, Z -6.3333, A 0.000, B 0.000, C 0.000 }
gfCNCPoint5[3131] = {X 429.8811, Y 25.9066, Z -6.3333, A 0.000, B 0.000, C 0.000 }
gfCNCPoint5[3132] = {X 429.4500, Y 24.0604, Z -6.3333, A 0.000, B 0.000, C 0.000 }
gfCNCPoint5[3133] = {X 429.2329, Y 22.1770, Z -6.3333, A 0.000, B 0.000, C 0.000 }
gfCNCPoint5[3134] = {X 429.2327, Y 20.2811, Z -6.3333, A 0.000, B 0.000, C 0.000 }
gfCNCPoint5[3135] = {X 429.4494, Y 18.3976, Z -6.3333, A 0.000, B 0.000, C 0.000 }
gfCNCPoint5[3136] = {X 429.8800, Y 16.5513, Z -6.3333, A 0.000, B 0.000, C 0.000 }
gfCNCPoint5[3137] = {X 430.4498, Y 15.0201, Z -6.3333, A 0.000, B 0.000, C 0.000 }
gfCNCPoint5[3138] = {X 431.2251, Y 13.5820, Z -6.3333, A 0.000, B 0.000, C 0.000 }
gfCNCPoint5[3139] = {X 432.1911, Y 12.2644, Z -6.3333, A 0.000, B 0.000, C 0.000 }
gfCNCPoint5[3140] = {X 433.3295, Y 11.0925, Z -6.3333, A 0.000, B 0.000, C 0.000 }
gfCNCPoint5[3141] = {X 434.6184, Y 10.0886, Z -6.3333, A 0.000, B 0.000, C 0.000 }
gfCNCPoint5[3142] = {X 436.0334, Y 9.2719, Z -6.3333, A 0.000, B 0.000, C 0.000 }
gfCNCPoint5[3143] = {X 437.5475, Y 8.6580, Z -6.3333, A 0.000, B 0.000, C 0.000 }
gfCNCPoint5[3144] = {X 439.1316, Y 8.2585, Z -6.3333, A 0.000, B 0.000, C 0.000 }
gfCNCPoint5[3145] = {X 441.2286, Y 7.9681, Z -6.3333, A 0.000, B 0.000, C 0.000 }
gfCNCPoint5[3146] = {X 443.3436, Y 7.8740, Z -6.3333, A 0.000, B 0.000, C 0.000 }
gfCNCPoint5[3147] = {X 444.0357, Y 7.8699, Z -6.3333, A 0.000, B 0.000, C 0.000 }
gfCNCPoint5[3148] = {X 459.4468, Y 7.8699, Z -6.3333, A 0.000, B 0.000, C 0.000 }
gfCNCPoint5[3149] = {X 460.4061, Y 7.9780, Z -6.3333, A 0.000, B 0.000, C 0.000 }
gfCNCPoint5[3150] = {X 461.3173, Y 8.2968, Z -6.3333, A 0.000, B 0.000, C 0.000 }
gfCNCPoint5[3151] = {X 462.1348, Y 8.8105, Z -6.3333, A 0.000, B 0.000, C 0.000 }
gfCNCPoint5[3152] = {X 462.8174, Y 9.4931, Z -6.3333, A 0.000, B 0.000, C 0.000 }
gfCNCPoint5[3153] = {X 463.3310, Y 10.3105, Z -6.3333, A 0.000, B 0.000, C 0.000 }
gfCNCPoint5[3154] = {X 463.6499, Y 11.2217, Z -6.3333, A 0.000, B 0.000, C 0.000 }
gfCNCPoint5[3155] = {X 463.7579, Y 12.1810, Z -6.3333, A 0.000, B 0.000, C 0.000 }
gfCNCPoint5[3156] = {X 463.7579, Y 12.9782, Z -6.3333, A 0.000, B 0.000, C 0.000 }
gfCNCPoint5[3157] = {X 463.6566, Y 13.9078, Z -6.3333, A 0.000, B 0.000, C 0.000 }
gfCNCPoint5[3158] = {X 463.3576, Y 14.7938, Z -6.3333, A 0.000, B 0.000, C 0.000 }
gfCNCPoint5[3159] = {X 462.8749, Y 15.5947, Z -6.3333, A 0.000, B 0.000, C 0.000 }
gfCNCPoint5[3160] = {X 462.2312, Y 16.2730, Z -6.3333, A 0.000, B 0.000, C 0.000 }
gfCNCPoint5[3161] = {X 462.2314, Y 28.5935, Z -6.3333, A 0.000, B 0.000, C 0.000 }
gfCNCPoint5[3162] = {X 466.2314, Y 28.5934, Z -6.3333, A 0.000, B 0.000, C 0.000 }
gfCNCPoint5[3163] = {X 462.1514, Y 28.5935, Z -6.3333, A 0.000, B 0.000, C 0.000 }
gfCNCPoint5[3164] = {X 462.1517, Y 40.9517, Z -6.3333, A 0.000, B 0.000, C 0.000 }
gfCNCPoint5[3165] = {X 462.1887, Y 40.9822, Z -6.3333, A 0.000, B 0.000, C 0.000 }
gfCNCPoint5[3166] = {X 462.8114, Y 41.6402, Z -6.3333, A 0.000, B 0.000, C 0.000 }
gfCNCPoint5[3167] = {X 463.2800, Y 42.4155, Z -6.3333, A 0.000, B 0.000, C 0.000 }
gfCNCPoint5[3168] = {X 463.5733, Y 43.2726, Z -6.3333, A 0.000, B 0.000, C 0.000 }
gfCNCPoint5[3169] = {X 463.6778, Y 44.1724, Z -6.3333, A 0.000, B 0.000, C 0.000 }
gfCNCPoint5[3170] = {X 463.6779, Y 45.0000, Z -6.3333, A 0.000, B 0.000, C 0.000 }
gfCNCPoint5[3171] = {X 463.5716, Y 45.9435, Z -6.3333, A 0.000, B 0.000, C 0.000 }
gfCNCPoint5[3172] = {X 463.2580, Y 46.8397, Z -6.3333, A 0.000, B 0.000, C 0.000 }
gfCNCPoint5[3173] = {X 462.7529, Y 47.6436, Z -6.3333, A 0.000, B 0.000, C 0.000 }
gfCNCPoint5[3174] = {X 462.0815, Y 48.3150, Z -6.3333, A 0.000, B 0.000, C 0.000 }
gfCNCPoint5[3175] = {X 461.2776, Y 48.8201, Z -6.3333, A 0.000, B 0.000, C 0.000 }
gfCNCPoint5[3176] = {X 460.3814, Y 49.1337, Z -6.3333, A 0.000, B 0.000, C 0.000 }
gfCNCPoint5[3177] = {X 459.4379, Y 49.2400, Z -6.3333, A 0.000, B 0.000, C 0.000 }
gfCNCPoint5[3178] = {X 452.9945, Y 49.2400, Z -6.3333, A 0.000, B 0.000, C 0.000 }
gfCNCPoint5[3179] = {X 452.0558, Y 49.1348, Z -6.3333, A 0.000, B 0.000, C 0.000 }
gfCNCPoint5[3180] = {X 451.1636, Y 48.8243, Z -6.3333, A 0.000, B 0.000, C 0.000 }
gfCNCPoint5[3181] = {X 450.3624, Y 48.3241, Z -6.3333, A 0.000, B 0.000, C 0.000 }
gfCNCPoint5[3182] = {X 449.6918, Y 47.6589, Z -6.3333, A 0.000, B 0.000, C 0.000 }
gfCNCPoint5[3183] = {X 449.1851, Y 46.8617, Z -6.3333, A 0.000, B 0.000, C 0.000 }
gfCNCPoint5[3184] = {X 448.8674, Y 45.9721, Z -6.3333, A 0.000, B 0.000, C 0.000 }
gfCNCPoint5[3185] = {X 448.7546, Y 45.0343, Z -6.3333, A 0.000, B 0.000, C 0.000 }
gfCNCPoint5[3186] = {X 448.7549, Y 44.1505, Z -6.3333, A 0.000, B 0.000, C 0.000 }
gfCNCPoint5[3187] = {X 448.8654, Y 43.2454, Z -6.3333, A 0.000, B 0.000, C 0.000 }
gfCNCPoint5[3188] = {X 449.1668, Y 42.3850, Z -6.3333, A 0.000, B 0.000, C 0.000 }
gfCNCPoint5[3189] = {X 449.6452, Y 41.6088, Z -6.3333, A 0.000, B 0.000, C 0.000 }
gfCNCPoint5[3190] = {X 450.2784, Y 40.9529, Z -6.3333, A 0.000, B 0.000, C 0.000 }
gfCNCPoint5[3191] = {X 450.2784, Y 34.3938, Z -6.3333, A 0.000, B 0.000, C 0.000 }
gfCNCPoint5[3192] = {X 447.4264, Y 34.3938, Z -6.3333, A 0.000, B 0.000, C 0.000 }
gfCNCPoint5[3193] = {X 443.1029, Y 42.8119, Z -6.3333, A 0.000, B 0.000, C 0.000 }
gfCNCPoint5[3194] = {X 443.1193, Y 42.8572, Z -6.3333, A 0.000, B 0.000, C 0.000 }
gfCNCPoint5[3195] = {X 443.2817, Y 43.5054, Z -6.3333, A 0.000, B 0.000, C 0.000 }
gfCNCPoint5[3196] = {X 443.3403, Y 44.1710, Z -6.3333, A 0.000, B 0.000, C 0.000 }
gfCNCPoint5[3197] = {X 443.3405, Y 45.0000, Z -6.3333, A 0.000, B 0.000, C 0.000 }
gfCNCPoint5[3198] = {X 443.2342, Y 45.9435, Z -6.3333, A 0.000, B 0.000, C 0.000 }
gfCNCPoint5[3199] = {X 442.9206, Y 46.8397, Z -6.3333, A 0.000, B 0.000, C 0.000 }
gfCNCPoint5[3200] = {X 442.4154, Y 47.6436, Z -6.3333, A 0.000, B 0.000, C 0.000 }
gfCNCPoint5[3201] = {X 441.7441, Y 48.3150, Z -6.3333, A 0.000, B 0.000, C 0.000 }
gfCNCPoint5[3202] = {X 440.9401, Y 48.8201, Z -6.3333, A 0.000, B 0.000, C 0.000 }
gfCNCPoint5[3203] = {X 440.0440, Y 49.1337, Z -6.3333, A 0.000, B 0.000, C 0.000 }
gfCNCPoint5[3204] = {X 439.1005, Y 49.2400, Z -6.3333, A 0.000, B 0.000, C 0.000 }
gfCNCPoint5[3205] = {X 432.5144, Y 49.2400, Z -6.3333, A 0.000, B 0.000, C 0.000 }
gfCNCPoint5[3206] = {X 431.5709, Y 49.1337, Z -6.3333, A 0.000, B 0.000, C 0.000 }
gfCNCPoint5[3207] = {X 430.6748, Y 48.8201, Z -6.3333, A 0.000, B 0.000, C 0.000 }
gfCNCPoint5[3208] = {X 429.8708, Y 48.3150, Z -6.3333, A 0.000, B 0.000, C 0.000 }
gfCNCPoint5[3209] = {X 429.1995, Y 47.6436, Z -6.3333, A 0.000, B 0.000, C 0.000 }
gfCNCPoint5[3210] = {X 428.6943, Y 46.8397, Z -6.3333, A 0.000, B 0.000, C 0.000 }
gfCNCPoint5[3211] = {X 428.3807, Y 45.9436, Z -6.3333, A 0.000, B 0.000, C 0.000 }
gfCNCPoint5[3212] = {X 428.2744, Y 45.0001, Z -6.3333, A 0.000, B 0.000, C 0.000 }
gfCNCPoint5[3213] = {X 428.2748, Y 44.1505, Z -6.3333, A 0.000, B 0.000, C 0.000 }
gfCNCPoint5[3214] = {X 428.3718, Y 43.3054, Z -6.3333, A 0.000, B 0.000, C 0.000 }
gfCNCPoint5[3215] = {X 428.6354, Y 42.4967, Z -6.3333, A 0.000, B 0.000, C 0.000 }
gfCNCPoint5[3216] = {X 429.0552, Y 41.7570, Z -6.3333, A 0.000, B 0.000, C 0.000 }
gfCNCPoint5[3217] = {X 429.6142, Y 41.1158, Z -6.3333, A 0.000, B 0.000, C 0.000 }
gfCNCPoint5[3218] = {X 430.2899, Y 40.5992, Z -6.3333, A 0.000, B 0.000, C 0.000 }
gfCNCPoint5[3219] = {X 431.0551, Y 40.2278, Z -6.3333, A 0.000, B 0.000, C 0.000 }
gfCNCPoint5[3220] = {X 435.0925, Y 32.3250, Z -6.3333, A 0.000, B 0.000, C 0.000 }
gfCNCPoint5[3221] = {X 433.9214, Y 31.5491, Z -6.3333, A 0.000, B 0.000, C 0.000 }
gfCNCPoint5[3222] = {X 432.8562, Y 30.6331, Z -6.3333, A 0.000, B 0.000, C 0.000 }
gfCNCPoint5[3223] = {X 431.9136, Y 29.5915, Z -6.3333, A 0.000, B 0.000, C 0.000 }
gfCNCPoint5[3224] = {X 431.1083, Y 28.4404, Z -6.3333, A 0.000, B 0.000, C 0.000 }
gfCNCPoint5[3225] = {X 430.4529, Y 27.1978, Z -6.3333, A 0.000, B 0.000, C 0.000 }
gfCNCPoint5[3226] = {X 429.9575, Y 25.8831, Z -6.3333, A 0.000, B 0.000, C 0.000 }
gfCNCPoint5[3227] = {X 429.5287, Y 24.0460, Z -6.3333, A 0.000, B 0.000, C 0.000 }
gfCNCPoint5[3228] = {X 429.3127, Y 22.1719, Z -6.3333, A 0.000, B 0.000, C 0.000 }
gfCNCPoint5[3229] = {X 429.3126, Y 20.2853, Z -6.3333, A 0.000, B 0.000, C 0.000 }
gfCNCPoint5[3230] = {X 429.5282, Y 18.4111, Z -6.3333, A 0.000, B 0.000, C 0.000 }
gfCNCPoint5[3231] = {X 429.9568, Y 16.5739, Z -6.3333, A 0.000, B 0.000, C 0.000 }
gfCNCPoint5[3232] = {X 430.5227, Y 15.0530, Z -6.3333, A 0.000, B 0.000, C 0.000 }
gfCNCPoint5[3233] = {X 431.2927, Y 13.6246, Z -6.3333, A 0.000, B 0.000, C 0.000 }
gfCNCPoint5[3234] = {X 432.2523, Y 12.3159, Z -6.3333, A 0.000, B 0.000, C 0.000 }
gfCNCPoint5[3235] = {X 433.3830, Y 11.1520, Z -6.3333, A 0.000, B 0.000, C 0.000 }
gfCNCPoint5[3236] = {X 434.6633, Y 10.1549, Z -6.3333, A 0.000, B 0.000, C 0.000 }
gfCNCPoint5[3237] = {X 436.0687, Y 9.3437, Z -6.3333, A 0.000, B 0.000, C 0.000 }
gfCNCPoint5[3238] = {X 437.5726, Y 8.7339, Z -6.3333, A 0.000, B 0.000, C 0.000 }
gfCNCPoint5[3239] = {X 439.1461, Y 8.3372, Z -6.3333, A 0.000, B 0.000, C 0.000 }
gfCNCPoint5[3240] = {X 441.2360, Y 8.0477, Z -6.3333, A 0.000, B 0.000, C 0.000 }
gfCNCPoint5[3241] = {X 443.3437, Y 7.9540, Z -6.3333, A 0.000, B 0.000, C 0.000 }
gfCNCPoint5[3242] = {X 444.0360, Y 7.9499, Z -6.3333, A 0.000, B 0.000, C 0.000 }
gfCNCPoint5[3243] = {X 459.4468, Y 7.9499, Z -6.3333, A 0.000, B 0.000, C 0.000 }
gfCNCPoint5[3244] = {X 460.3883, Y 8.0560, Z -6.3333, A 0.000, B 0.000, C 0.000 }
gfCNCPoint5[3245] = {X 461.2826, Y 8.3689, Z -6.3333, A 0.000, B 0.000, C 0.000 }
gfCNCPoint5[3246] = {X 462.0849, Y 8.8730, Z -6.3333, A 0.000, B 0.000, C 0.000 }
gfCNCPoint5[3247] = {X 462.7548, Y 9.5430, Z -6.3333, A 0.000, B 0.000, C 0.000 }
gfCNCPoint5[3248] = {X 463.2589, Y 10.3452, Z -6.3333, A 0.000, B 0.000, C 0.000 }
gfCNCPoint5[3249] = {X 463.5719, Y 11.2395, Z -6.3333, A 0.000, B 0.000, C 0.000 }
gfCNCPoint5[3250] = {X 463.6779, Y 12.1810, Z -6.3333, A 0.000, B 0.000, C 0.000 }
gfCNCPoint5[3251] = {X 463.6779, Y 12.9782, Z -6.3333, A 0.000, B 0.000, C 0.000 }
gfCNCPoint5[3252] = {X 463.5765, Y 13.8996, Z -6.3333, A 0.000, B 0.000, C 0.000 }
gfCNCPoint5[3253] = {X 463.2772, Y 14.7769, Z -6.3333, A 0.000, B 0.000, C 0.000 }
gfCNCPoint5[3254] = {X 462.7944, Y 15.5683, Z -6.3333, A 0.000, B 0.000, C 0.000 }
gfCNCPoint5[3255] = {X 462.1512, Y 16.2358, Z -6.3333, A 0.000, B 0.000, C 0.000 }
gfCNCPoint5[3256] = {X 462.1514, Y 28.5935, Z -6.3333, A 0.000, B 0.000, C 0.000 }
gfCNCPoint5[3257] = {X 466.1514, Y 28.5934, Z -6.3333, A 0.000, B 0.000, C 0.000 }
gfCNCPoint5[3258] = {X 462.0714, Y 28.5935, Z -6.3333, A 0.000, B 0.000, C 0.000 }
gfCNCPoint5[3259] = {X 462.0717, Y 40.9895, Z -6.3333, A 0.000, B 0.000, C 0.000 }
gfCNCPoint5[3260] = {X 462.1373, Y 41.0435, Z -6.3333, A 0.000, B 0.000, C 0.000 }
gfCNCPoint5[3261] = {X 462.7480, Y 41.6891, Z -6.3333, A 0.000, B 0.000, C 0.000 }
gfCNCPoint5[3262] = {X 463.2077, Y 42.4496, Z -6.3333, A 0.000, B 0.000, C 0.000 }
gfCNCPoint5[3263] = {X 463.4953, Y 43.2904, Z -6.3333, A 0.000, B 0.000, C 0.000 }
gfCNCPoint5[3264] = {X 463.5978, Y 44.1731, Z -6.3333, A 0.000, B 0.000, C 0.000 }
gfCNCPoint5[3265] = {X 463.5979, Y 45.0000, Z -6.3333, A 0.000, B 0.000, C 0.000 }
gfCNCPoint5[3266] = {X 463.4936, Y 45.9257, Z -6.3333, A 0.000, B 0.000, C 0.000 }
gfCNCPoint5[3267] = {X 463.1860, Y 46.8050, Z -6.3333, A 0.000, B 0.000, C 0.000 }
gfCNCPoint5[3268] = {X 462.6904, Y 47.5937, Z -6.3333, A 0.000, B 0.000, C 0.000 }
gfCNCPoint5[3269] = {X 462.0317, Y 48.2524, Z -6.3333, A 0.000, B 0.000, C 0.000 }
gfCNCPoint5[3270] = {X 461.2429, Y 48.7480, Z -6.3333, A 0.000, B 0.000, C 0.000 }
gfCNCPoint5[3271] = {X 460.3636, Y 49.0557, Z -6.3333, A 0.000, B 0.000, C 0.000 }
gfCNCPoint5[3272] = {X 459.4379, Y 49.1600, Z -6.3333, A 0.000, B 0.000, C 0.000 }
gfCNCPoint5[3273] = {X 452.9945, Y 49.1600, Z -6.3333, A 0.000, B 0.000, C 0.000 }
gfCNCPoint5[3274] = {X 452.0735, Y 49.0568, Z -6.3333, A 0.000, B 0.000, C 0.000 }
gfCNCPoint5[3275] = {X 451.1982, Y 48.7522, Z -6.3333, A 0.000, B 0.000, C 0.000 }
gfCNCPoint5[3276] = {X 450.4120, Y 48.2614, Z -6.3333, A 0.000, B 0.000, C 0.000 }
gfCNCPoint5[3277] = {X 449.7541, Y 47.6087, Z -6.3333, A 0.000, B 0.000, C 0.000 }
gfCNCPoint5[3278] = {X 449.2569, Y 46.8266, Z -6.3333, A 0.000, B 0.000, C 0.000 }
gfCNCPoint5[3279] = {X 448.9453, Y 45.9538, Z -6.3333, A 0.000, B 0.000, C 0.000 }
gfCNCPoint5[3280] = {X 448.8346, Y 45.0336, Z -6.3333, A 0.000, B 0.000, C 0.000 }
gfCNCPoint5[3281] = {X 448.8349, Y 44.1516, Z -6.3333, A 0.000, B 0.000, C 0.000 }
gfCNCPoint5[3282] = {X 448.9454, Y 43.2545, Z -6.3333, A 0.000, B 0.000, C 0.000 }
gfCNCPoint5[3283] = {X 449.2471, Y 42.4026, Z -6.3333, A 0.000, B 0.000, C 0.000 }
gfCNCPoint5[3284] = {X 449.7256, Y 41.6358, Z -6.3333, A 0.000, B 0.000, C 0.000 }
gfCNCPoint5[3285] = {X 450.3584, Y 40.9906, Z -6.3333, A 0.000, B 0.000, C 0.000 }
gfCNCPoint5[3286] = {X 450.3584, Y 34.3138, Z -6.3333, A 0.000, B 0.000, C 0.000 }
gfCNCPoint5[3287] = {X 447.3776, Y 34.3138, Z -6.3333, A 0.000, B 0.000, C 0.000 }
gfCNCPoint5[3288] = {X 443.0158, Y 42.8063, Z -6.3333, A 0.000, B 0.000, C 0.000 }
gfCNCPoint5[3289] = {X 443.0437, Y 42.8836, Z -6.3333, A 0.000, B 0.000, C 0.000 }
gfCNCPoint5[3290] = {X 443.2029, Y 43.5191, Z -6.3333, A 0.000, B 0.000, C 0.000 }
gfCNCPoint5[3291] = {X 443.2603, Y 44.1717, Z -6.3333, A 0.000, B 0.000, C 0.000 }
gfCNCPoint5[3292] = {X 443.2605, Y 45.0000, Z -6.3333, A 0.000, B 0.000, C 0.000 }
gfCNCPoint5[3293] = {X 443.1562, Y 45.9257, Z -6.3333, A 0.000, B 0.000, C 0.000 }
gfCNCPoint5[3294] = {X 442.8485, Y 46.8050, Z -6.3333, A 0.000, B 0.000, C 0.000 }
gfCNCPoint5[3295] = {X 442.3529, Y 47.5937, Z -6.3333, A 0.000, B 0.000, C 0.000 }
gfCNCPoint5[3296] = {X 441.6942, Y 48.2524, Z -6.3333, A 0.000, B 0.000, C 0.000 }
gfCNCPoint5[3297] = {X 440.9054, Y 48.7480, Z -6.3333, A 0.000, B 0.000, C 0.000 }
gfCNCPoint5[3298] = {X 440.0262, Y 49.0557, Z -6.3333, A 0.000, B 0.000, C 0.000 }
gfCNCPoint5[3299] = {X 439.1005, Y 49.1600, Z -6.3333, A 0.000, B 0.000, C 0.000 }
gfCNCPoint5[3300] = {X 432.5144, Y 49.1600, Z -6.3333, A 0.000, B 0.000, C 0.000 }
gfCNCPoint5[3301] = {X 431.5887, Y 49.0557, Z -6.3333, A 0.000, B 0.000, C 0.000 }
gfCNCPoint5[3302] = {X 430.7095, Y 48.7480, Z -6.3333, A 0.000, B 0.000, C 0.000 }
gfCNCPoint5[3303] = {X 429.9207, Y 48.2524, Z -6.3333, A 0.000, B 0.000, C 0.000 }
gfCNCPoint5[3304] = {X 429.2620, Y 47.5937, Z -6.3333, A 0.000, B 0.000, C 0.000 }
gfCNCPoint5[3305] = {X 428.7664, Y 46.8050, Z -6.3333, A 0.000, B 0.000, C 0.000 }
gfCNCPoint5[3306] = {X 428.4587, Y 45.9257, Z -6.3333, A 0.000, B 0.000, C 0.000 }
gfCNCPoint5[3307] = {X 428.3544, Y 45.0000, Z -6.3333, A 0.000, B 0.000, C 0.000 }
gfCNCPoint5[3308] = {X 428.3548, Y 44.1516, Z -6.3333, A 0.000, B 0.000, C 0.000 }
gfCNCPoint5[3309] = {X 428.4510, Y 43.3174, Z -6.3333, A 0.000, B 0.000, C 0.000 }
gfCNCPoint5[3310] = {X 428.7128, Y 42.5195, Z -6.3333, A 0.000, B 0.000, C 0.000 }
gfCNCPoint5[3311] = {X 429.1295, Y 41.7905, Z -6.3333, A 0.000, B 0.000, C 0.000 }
gfCNCPoint5[3312] = {X 429.6841, Y 41.1600, Z -6.3333, A 0.000, B 0.000, C 0.000 }
gfCNCPoint5[3313] = {X 430.3541, Y 40.6537, Z -6.3333, A 0.000, B 0.000, C 0.000 }
gfCNCPoint5[3314] = {X 431.1120, Y 40.2923, Z -6.3333, A 0.000, B 0.000, C 0.000 }
gfCNCPoint5[3315] = {X 435.1985, Y 32.2934, Z -6.3333, A 0.000, B 0.000, C 0.000 }
gfCNCPoint5[3316] = {X 434.0203, Y 31.5234, Z -6.3333, A 0.000, B 0.000, C 0.000 }
gfCNCPoint5[3317] = {X 432.9484, Y 30.6112, Z -6.3333, A 0.000, B 0.000, C 0.000 }
gfCNCPoint5[3318] = {X 431.9999, Y 29.5713, Z -6.3333, A 0.000, B 0.000, C 0.000 }
gfCNCPoint5[3319] = {X 431.1898, Y 28.4203, Z -6.3333, A 0.000, B 0.000, C 0.000 }
gfCNCPoint5[3320] = {X 430.5310, Y 27.1765, Z -6.3333, A 0.000, B 0.000, C 0.000 }
gfCNCPoint5[3321] = {X 430.0340, Y 25.8597, Z -6.3333, A 0.000, B 0.000, C 0.000 }
gfCNCPoint5[3322] = {X 429.6074, Y 24.0316, Z -6.3333, A 0.000, B 0.000, C 0.000 }
gfCNCPoint5[3323] = {X 429.3926, Y 22.1667, Z -6.3333, A 0.000, B 0.000, C 0.000 }
gfCNCPoint5[3324] = {X 429.3925, Y 20.2895, Z -6.3333, A 0.000, B 0.000, C 0.000 }
gfCNCPoint5[3325] = {X 429.6071, Y 18.4246, Z -6.3333, A 0.000, B 0.000, C 0.000 }
gfCNCPoint5[3326] = {X 430.0335, Y 16.5965, Z -6.3333, A 0.000, B 0.000, C 0.000 }
gfCNCPoint5[3327] = {X 430.5956, Y 15.0860, Z -6.3333, A 0.000, B 0.000, C 0.000 }
gfCNCPoint5[3328] = {X 431.3604, Y 13.6673, Z -6.3333, A 0.000, B 0.000, C 0.000 }
gfCNCPoint5[3329] = {X 432.3135, Y 12.3675, Z -6.3333, A 0.000, B 0.000, C 0.000 }
gfCNCPoint5[3330] = {X 433.4365, Y 11.2114, Z -6.3333, A 0.000, B 0.000, C 0.000 }
gfCNCPoint5[3331] = {X 434.7081, Y 10.2211, Z -6.3333, A 0.000, B 0.000, C 0.000 }
gfCNCPoint5[3332] = {X 436.1040, Y 9.4155, Z -6.3333, A 0.000, B 0.000, C 0.000 }
gfCNCPoint5[3333] = {X 437.5977, Y 8.8099, Z -6.3333, A 0.000, B 0.000, C 0.000 }
gfCNCPoint5[3334] = {X 439.1605, Y 8.4159, Z -6.3333, A 0.000, B 0.000, C 0.000 }
gfCNCPoint5[3335] = {X 441.2433, Y 8.1274, Z -6.3333, A 0.000, B 0.000, C 0.000 }
gfCNCPoint5[3336] = {X 443.3439, Y 8.0340, Z -6.3333, A 0.000, B 0.000, C 0.000 }
gfCNCPoint5[3337] = {X 444.0362, Y 8.0299, Z -6.3333, A 0.000, B 0.000, C 0.000 }
gfCNCPoint5[3338] = {X 459.4468, Y 8.0299, Z -6.3333, A 0.000, B 0.000, C 0.000 }
gfCNCPoint5[3339] = {X 460.3705, Y 8.1340, Z -6.3333, A 0.000, B 0.000, C 0.000 }
gfCNCPoint5[3340] = {X 461.2479, Y 8.4410, Z -6.3333, A 0.000, B 0.000, C 0.000 }
gfCNCPoint5[3341] = {X 462.0350, Y 8.9355, Z -6.3333, A 0.000, B 0.000, C 0.000 }
gfCNCPoint5[3342] = {X 462.6923, Y 9.5928, Z -6.3333, A 0.000, B 0.000, C 0.000 }
gfCNCPoint5[3343] = {X 463.1869, Y 10.3799, Z -6.3333, A 0.000, B 0.000, C 0.000 }
gfCNCPoint5[3344] = {X 463.4939, Y 11.2573, Z -6.3333, A 0.000, B 0.000, C 0.000 }
gfCNCPoint5[3345] = {X 463.5979, Y 12.1810, Z -6.3333, A 0.000, B 0.000, C 0.000 }
gfCNCPoint5[3346] = {X 463.5979, Y 12.9782, Z -6.3333, A 0.000, B 0.000, C 0.000 }
gfCNCPoint5[3347] = {X 463.5023, Y 13.8649, Z -6.3333, A 0.000, B 0.000, C 0.000 }
gfCNCPoint5[3348] = {X 463.2198, Y 14.7109, Z -6.3333, A 0.000, B 0.000, C 0.000 }
gfCNCPoint5[3349] = {X 462.7636, Y 15.4772, Z -6.3333, A 0.000, B 0.000, C 0.000 }
gfCNCPoint5[3350] = {X 462.1544, Y 16.1287, Z -6.3333, A 0.000, B 0.000, C 0.000 }
gfCNCPoint5[3351] = {X 462.0712, Y 16.1985, Z -6.3333, A 0.000, B 0.000, C 0.000 }
gfCNCPoint5[3352] = {X 462.0714, Y 28.5935, Z -6.3333, A 0.000, B 0.000, C 0.000 }
gfCNCPoint5[3353] = {X 466.0714, Y 28.5934, Z -6.3333, A 0.000, B 0.000, C 0.000 }
gfCNCPoint5[3354] = {X 461.9914, Y 28.5935, Z -6.3333, A 0.000, B 0.000, C 0.000 }
gfCNCPoint5[3355] = {X 461.9917, Y 41.0273, Z -6.3333, A 0.000, B 0.000, C 0.000 }
gfCNCPoint5[3356] = {X 462.0860, Y 41.1049, Z -6.3333, A 0.000, B 0.000, C 0.000 }
gfCNCPoint5[3357] = {X 462.6847, Y 41.7380, Z -6.3333, A 0.000, B 0.000, C 0.000 }
gfCNCPoint5[3358] = {X 463.1353, Y 42.4838, Z -6.3333, A 0.000, B 0.000, C 0.000 }
gfCNCPoint5[3359] = {X 463.4173, Y 43.3083, Z -6.3333, A 0.000, B 0.000, C 0.000 }
gfCNCPoint5[3360] = {X 463.5178, Y 44.1738, Z -6.3333, A 0.000, B 0.000, C 0.000 }
gfCNCPoint5[3361] = {X 463.5179, Y 45.0000, Z -6.3333, A 0.000, B 0.000, C 0.000 }
gfCNCPoint5[3362] = {X 463.4156, Y 45.9079, Z -6.3333, A 0.000, B 0.000, C 0.000 }
gfCNCPoint5[3363] = {X 463.1139, Y 46.7702, Z -6.3333, A 0.000, B 0.000, C 0.000 }
gfCNCPoint5[3364] = {X 462.6278, Y 47.5438, Z -6.3333, A 0.000, B 0.000, C 0.000 }
gfCNCPoint5[3365] = {X 461.9818, Y 48.1899, Z -6.3333, A 0.000, B 0.000, C 0.000 }
gfCNCPoint5[3366] = {X 461.2082, Y 48.6760, Z -6.3333, A 0.000, B 0.000, C 0.000 }
gfCNCPoint5[3367] = {X 460.3458, Y 48.9777, Z -6.3333, A 0.000, B 0.000, C 0.000 }
gfCNCPoint5[3368] = {X 459.4379, Y 49.0800, Z -6.3333, A 0.000, B 0.000, C 0.000 }
gfCNCPoint5[3369] = {X 452.9945, Y 49.0800, Z -6.3333, A 0.000, B 0.000, C 0.000 }
gfCNCPoint5[3370] = {X 452.0912, Y 48.9788, Z -6.3333, A 0.000, B 0.000, C 0.000 }
gfCNCPoint5[3371] = {X 451.2327, Y 48.6800, Z -6.3333, A 0.000, B 0.000, C 0.000 }
gfCNCPoint5[3372] = {X 450.4617, Y 48.1987, Z -6.3333, A 0.000, B 0.000, C 0.000 }
gfCNCPoint5[3373] = {X 449.8164, Y 47.5585, Z -6.3333, A 0.000, B 0.000, C 0.000 }
gfCNCPoint5[3374] = {X 449.3288, Y 46.7914, Z -6.3333, A 0.000, B 0.000, C 0.000 }
gfCNCPoint5[3375] = {X 449.0232, Y 45.9354, Z -6.3333, A 0.000, B 0.000, C 0.000 }
gfCNCPoint5[3376] = {X 448.9146, Y 45.0330, Z -6.3333, A 0.000, B 0.000, C 0.000 }
gfCNCPoint5[3377] = {X 448.9149, Y 44.1527, Z -6.3333, A 0.000, B 0.000, C 0.000 }
gfCNCPoint5[3378] = {X 449.0254, Y 43.2637, Z -6.3333, A 0.000, B 0.000, C 0.000 }
gfCNCPoint5[3379] = {X 449.3274, Y 42.4203, Z -6.3333, A 0.000, B 0.000, C 0.000 }
gfCNCPoint5[3380] = {X 449.8061, Y 41.6631, Z -6.3333, A 0.000, B 0.000, C 0.000 }
gfCNCPoint5[3381] = {X 450.4384, Y 41.0287, Z -6.3333, A 0.000, B 0.000, C 0.000 }
gfCNCPoint5[3382] = {X 450.4384, Y 34.2338, Z -6.3333, A 0.000, B 0.000, C 0.000 }
gfCNCPoint5[3383] = {X 447.3287, Y 34.2338, Z -6.3333, A 0.000, B 0.000, C 0.000 }
gfCNCPoint5[3384] = {X 442.9287, Y 42.8007, Z -6.3333, A 0.000, B 0.000, C 0.000 }
gfCNCPoint5[3385] = {X 442.9682, Y 42.9099, Z -6.3333, A 0.000, B 0.000, C 0.000 }
gfCNCPoint5[3386] = {X 443.1241, Y 43.5328, Z -6.3333, A 0.000, B 0.000, C 0.000 }
gfCNCPoint5[3387] = {X 443.1803, Y 44.1725, Z -6.3333, A 0.000, B 0.000, C 0.000 }
gfCNCPoint5[3388] = {X 443.1805, Y 45.0000, Z -6.3333, A 0.000, B 0.000, C 0.000 }
gfCNCPoint5[3389] = {X 443.0782, Y 45.9079, Z -6.3333, A 0.000, B 0.000, C 0.000 }
gfCNCPoint5[3390] = {X 442.7764, Y 46.7702, Z -6.3333, A 0.000, B 0.000, C 0.000 }
gfCNCPoint5[3391] = {X 442.2903, Y 47.5438, Z -6.3333, A 0.000, B 0.000, C 0.000 }
gfCNCPoint5[3392] = {X 441.6443, Y 48.1899, Z -6.3333, A 0.000, B 0.000, C 0.000 }
gfCNCPoint5[3393] = {X 440.8707, Y 48.6760, Z -6.3333, A 0.000, B 0.000, C 0.000 }
gfCNCPoint5[3394] = {X 440.0084, Y 48.9777, Z -6.3333, A 0.000, B 0.000, C 0.000 }
gfCNCPoint5[3395] = {X 439.1005, Y 49.0800, Z -6.3333, A 0.000, B 0.000, C 0.000 }
gfCNCPoint5[3396] = {X 432.5144, Y 49.0800, Z -6.3333, A 0.000, B 0.000, C 0.000 }
gfCNCPoint5[3397] = {X 431.6065, Y 48.9777, Z -6.3333, A 0.000, B 0.000, C 0.000 }
gfCNCPoint5[3398] = {X 430.7442, Y 48.6760, Z -6.3333, A 0.000, B 0.000, C 0.000 }
gfCNCPoint5[3399] = {X 429.9706, Y 48.1899, Z -6.3333, A 0.000, B 0.000, C 0.000 }
gfCNCPoint5[3400] = {X 429.3245, Y 47.5438, Z -6.3333, A 0.000, B 0.000, C 0.000 }
gfCNCPoint5[3401] = {X 428.8385, Y 46.7702, Z -6.3333, A 0.000, B 0.000, C 0.000 }
gfCNCPoint5[3402] = {X 428.5367, Y 45.9079, Z -6.3333, A 0.000, B 0.000, C 0.000 }
gfCNCPoint5[3403] = {X 428.4344, Y 45.0000, Z -6.3333, A 0.000, B 0.000, C 0.000 }
gfCNCPoint5[3404] = {X 428.4348, Y 44.1527, Z -6.3333, A 0.000, B 0.000, C 0.000 }
gfCNCPoint5[3405] = {X 428.5303, Y 43.3294, Z -6.3333, A 0.000, B 0.000, C 0.000 }
gfCNCPoint5[3406] = {X 428.7902, Y 42.5424, Z -6.3333, A 0.000, B 0.000, C 0.000 }
gfCNCPoint5[3407] = {X 429.2038, Y 41.8242, Z -6.3333, A 0.000, B 0.000, C 0.000 }
gfCNCPoint5[3408] = {X 429.7540, Y 41.2044, Z -6.3333, A 0.000, B 0.000, C 0.000 }
gfCNCPoint5[3409] = {X 430.4181, Y 40.7085, Z -6.3333, A 0.000, B 0.000, C 0.000 }
gfCNCPoint5[3410] = {X 431.1687, Y 40.3571, Z -6.3333, A 0.000, B 0.000, C 0.000 }
gfCNCPoint5[3411] = {X 435.3047, Y 32.2613, Z -6.3333, A 0.000, B 0.000, C 0.000 }
gfCNCPoint5[3412] = {X 434.1195, Y 31.4974, Z -6.3333, A 0.000, B 0.000, C 0.000 }
gfCNCPoint5[3413] = {X 433.0408, Y 30.5890, Z -6.3333, A 0.000, B 0.000, C 0.000 }
gfCNCPoint5[3414] = {X 432.0863, Y 29.5510, Z -6.3333, A 0.000, B 0.000, C 0.000 }
gfCNCPoint5[3415] = {X 431.2714, Y 28.4002, Z -6.3333, A 0.000, B 0.000, C 0.000 }
gfCNCPoint5[3416] = {X 430.6092, Y 27.1552, Z -6.3333, A 0.000, B 0.000, C 0.000 }
gfCNCPoint5[3417] = {X 430.1105, Y 25.8362, Z -6.3333, A 0.000, B 0.000, C 0.000 }
gfCNCPoint5[3418] = {X 429.6861, Y 24.0172, Z -6.3333, A 0.000, B 0.000, C 0.000 }
gfCNCPoint5[3419] = {X 429.4724, Y 22.1616, Z -6.3333, A 0.000, B 0.000, C 0.000 }
gfCNCPoint5[3420] = {X 429.4724, Y 20.2937, Z -6.3333, A 0.000, B 0.000, C 0.000 }
gfCNCPoint5[3421] = {X 429.6859, Y 18.4381, Z -6.3333, A 0.000, B 0.000, C 0.000 }
gfCNCPoint5[3422] = {X 430.1102, Y 16.6191, Z -6.3333, A 0.000, B 0.000, C 0.000 }
gfCNCPoint5[3423] = {X 430.6685, Y 15.1189, Z -6.3333, A 0.000, B 0.000, C 0.000 }
gfCNCPoint5[3424] = {X 431.4281, Y 13.7099, Z -6.3333, A 0.000, B 0.000, C 0.000 }
gfCNCPoint5[3425] = {X 432.3746, Y 12.4190, Z -6.3333, A 0.000, B 0.000, C 0.000 }
gfCNCPoint5[3426] = {X 433.4900, Y 11.2709, Z -6.3333, A 0.000, B 0.000, C 0.000 }
gfCNCPoint5[3427] = {X 434.7529, Y 10.2874, Z -6.3333, A 0.000, B 0.000, C 0.000 }
gfCNCPoint5[3428] = {X 436.1393, Y 9.4873, Z -6.3333, A 0.000, B 0.000, C 0.000 }
gfCNCPoint5[3429] = {X 437.6227, Y 8.8859, Z -6.3333, A 0.000, B 0.000, C 0.000 }
gfCNCPoint5[3430] = {X 439.1749, Y 8.4945, Z -6.3333, A 0.000, B 0.000, C 0.000 }
gfCNCPoint5[3431] = {X 441.2506, Y 8.2071, Z -6.3333, A 0.000, B 0.000, C 0.000 }
gfCNCPoint5[3432] = {X 443.3440, Y 8.1140, Z -6.3333, A 0.000, B 0.000, C 0.000 }
gfCNCPoint5[3433] = {X 444.0364, Y 8.1099, Z -6.3333, A 0.000, B 0.000, C 0.000 }
gfCNCPoint5[3434] = {X 459.4468, Y 8.1099, Z -6.3333, A 0.000, B 0.000, C 0.000 }
gfCNCPoint5[3435] = {X 460.3527, Y 8.2120, Z -6.3333, A 0.000, B 0.000, C 0.000 }
gfCNCPoint5[3436] = {X 461.2132, Y 8.5131, Z -6.3333, A 0.000, B 0.000, C 0.000 }
gfCNCPoint5[3437] = {X 461.9851, Y 8.9981, Z -6.3333, A 0.000, B 0.000, C 0.000 }
gfCNCPoint5[3438] = {X 462.6297, Y 9.6427, Z -6.3333, A 0.000, B 0.000, C 0.000 }
gfCNCPoint5[3439] = {X 463.1148, Y 10.4146, Z -6.3333, A 0.000, B 0.000, C 0.000 }
gfCNCPoint5[3440] = {X 463.4159, Y 11.2751, Z -6.3333, A 0.000, B 0.000, C 0.000 }
gfCNCPoint5[3441] = {X 463.5179, Y 12.1810, Z -6.3333, A 0.000, B 0.000, C 0.000 }
gfCNCPoint5[3442] = {X 463.5179, Y 12.9782, Z -6.3333, A 0.000, B 0.000, C 0.000 }
gfCNCPoint5[3443] = {X 463.4241, Y 13.8478, Z -6.3333, A 0.000, B 0.000, C 0.000 }
gfCNCPoint5[3444] = {X 463.1471, Y 14.6776, Z -6.3333, A 0.000, B 0.000, C 0.000 }
gfCNCPoint5[3445] = {X 462.6996, Y 15.4291, Z -6.3333, A 0.000, B 0.000, C 0.000 }
gfCNCPoint5[3446] = {X 462.1022, Y 16.0681, Z -6.3333, A 0.000, B 0.000, C 0.000 }
gfCNCPoint5[3447] = {X 462.0446, Y 16.1168, Z -6.3333, A 0.000, B 0.000, C 0.000 }
gfCNCPoint5[3448] = {X 461.9861, Y 16.1644, Z -6.3333, A 0.000, B 0.000, C 0.000 }
gfCNCPoint5[3449] = {X 461.9912, Y 16.1985, Z -6.3333, A 0.000, B 0.000, C 0.000 }
gfCNCPoint5[3450] = {X 461.9914, Y 28.5935, Z -6.3333, A 0.000, B 0.000, C 0.000 }
gfCNCPoint5[3451] = {X 465.9914, Y 28.5934, Z -6.3333, A 0.000, B 0.000, C 0.000 }
gfCNCPoint5[3452] = {X 465.9914, Y 28.5933, Z -6.3333, A 0.000, B 0.000, C 0.000 }
gfCNCPoint5[3453] = {X 461.9111, Y 28.5935, Z -6.3333, A 0.000, B 0.000, C 0.000 }
gfCNCPoint5[3454] = {X 461.9117, Y 41.0651, Z -6.3333, A 0.000, B 0.000, C 0.000 }
gfCNCPoint5[3455] = {X 462.0504, Y 41.1798, Z -6.3333, A 0.000, B 0.000, C 0.000 }
gfCNCPoint5[3456] = {X 462.6360, Y 41.8062, Z -6.3333, A 0.000, B 0.000, C 0.000 }
gfCNCPoint5[3457] = {X 463.0746, Y 42.5430, Z -6.3333, A 0.000, B 0.000, C 0.000 }
gfCNCPoint5[3458] = {X 463.3460, Y 43.3563, Z -6.3333, A 0.000, B 0.000, C 0.000 }
gfCNCPoint5[3459] = {X 463.4379, Y 44.2088, Z -6.3333, A 0.000, B 0.000, C 0.000 }
gfCNCPoint5[3460] = {X 463.4379, Y 45.0000, Z -6.3333, A 0.000, B 0.000, C 0.000 }
gfCNCPoint5[3461] = {X 463.3377, Y 45.8901, Z -6.3333, A 0.000, B 0.000, C 0.000 }
gfCNCPoint5[3462] = {X 463.0418, Y 46.7355, Z -6.3333, A 0.000, B 0.000, C 0.000 }
gfCNCPoint5[3463] = {X 462.5653, Y 47.4940, Z -6.3333, A 0.000, B 0.000, C 0.000 }
gfCNCPoint5[3464] = {X 461.9319, Y 48.1273, Z -6.3333, A 0.000, B 0.000, C 0.000 }
gfCNCPoint5[3465] = {X 461.1735, Y 48.6039, Z -6.3333, A 0.000, B 0.000, C 0.000 }
gfCNCPoint5[3466] = {X 460.3280, Y 48.8997, Z -6.3333, A 0.000, B 0.000, C 0.000 }
gfCNCPoint5[3467] = {X 459.4379, Y 49.0000, Z -6.3333, A 0.000, B 0.000, C 0.000 }
gfCNCPoint5[3468] = {X 452.9945, Y 49.0000, Z -6.3333, A 0.000, B 0.000, C 0.000 }
gfCNCPoint5[3469] = {X 452.1044, Y 48.8997, Z -6.3333, A 0.000, B 0.000, C 0.000 }
gfCNCPoint5[3470] = {X 451.2589, Y 48.6039, Z -6.3333, A 0.000, B 0.000, C 0.000 }
gfCNCPoint5[3471] = {X 450.5005, Y 48.1273, Z -6.3333, A 0.000, B 0.000, C 0.000 }
gfCNCPoint5[3472] = {X 449.8671, Y 47.4939, Z -6.3333, A 0.000, B 0.000, C 0.000 }
gfCNCPoint5[3473] = {X 449.3906, Y 46.7355, Z -6.3333, A 0.000, B 0.000, C 0.000 }
gfCNCPoint5[3474] = {X 449.0948, Y 45.8901, Z -6.3333, A 0.000, B 0.000, C 0.000 }
gfCNCPoint5[3475] = {X 448.9945, Y 45.0000, Z -6.3333, A 0.000, B 0.000, C 0.000 }
gfCNCPoint5[3476] = {X 448.9949, Y 44.1538, Z -6.3333, A 0.000, B 0.000, C 0.000 }
gfCNCPoint5[3477] = {X 449.1055, Y 43.2730, Z -6.3333, A 0.000, B 0.000, C 0.000 }
gfCNCPoint5[3478] = {X 449.4077, Y 42.4382, Z -6.3333, A 0.000, B 0.000, C 0.000 }
gfCNCPoint5[3479] = {X 449.8865, Y 41.6907, Z -6.3333, A 0.000, B 0.000, C 0.000 }
gfCNCPoint5[3480] = {X 450.5184, Y 41.0672, Z -6.3333, A 0.000, B 0.000, C 0.000 }
gfCNCPoint5[3481] = {X 450.5184, Y 34.1538, Z -6.3333, A 0.000, B 0.000, C 0.000 }
gfCNCPoint5[3482] = {X 447.5241, Y 34.1538, Z -6.3333, A 0.000, B 0.000, C 0.000 }
gfCNCPoint5[3483] = {X 447.2799, Y 34.1538, Z -6.3333, A 0.000, B 0.000, C 0.000 }
gfCNCPoint5[3484] = {X 442.8416, Y 42.7952, Z -6.3333, A 0.000, B 0.000, C 0.000 }
gfCNCPoint5[3485] = {X 442.8971, Y 42.9495, Z -6.3333, A 0.000, B 0.000, C 0.000 }
gfCNCPoint5[3486] = {X 443.0493, Y 43.5710, Z -6.3333, A 0.000, B 0.000, C 0.000 }
gfCNCPoint5[3487] = {X 443.1005, Y 44.2089, Z -6.3333, A 0.000, B 0.000, C 0.000 }
gfCNCPoint5[3488] = {X 443.1005, Y 45.0000, Z -6.3333, A 0.000, B 0.000, C 0.000 }
gfCNCPoint5[3489] = {X 443.0002, Y 45.8901, Z -6.3333, A 0.000, B 0.000, C 0.000 }
gfCNCPoint5[3490] = {X 442.7043, Y 46.7355, Z -6.3333, A 0.000, B 0.000, C 0.000 }
gfCNCPoint5[3491] = {X 442.2278, Y 47.4940, Z -6.3333, A 0.000, B 0.000, C 0.000 }
gfCNCPoint5[3492] = {X 441.5944, Y 48.1273, Z -6.3333, A 0.000, B 0.000, C 0.000 }
gfCNCPoint5[3493] = {X 440.8360, Y 48.6039, Z -6.3333, A 0.000, B 0.000, C 0.000 }
gfCNCPoint5[3494] = {X 439.9906, Y 48.8997, Z -6.3333, A 0.000, B 0.000, C 0.000 }
gfCNCPoint5[3495] = {X 439.1005, Y 49.0000, Z -6.3333, A 0.000, B 0.000, C 0.000 }
gfCNCPoint5[3496] = {X 432.5144, Y 49.0000, Z -6.3333, A 0.000, B 0.000, C 0.000 }
gfCNCPoint5[3497] = {X 431.6243, Y 48.8997, Z -6.3333, A 0.000, B 0.000, C 0.000 }
gfCNCPoint5[3498] = {X 430.7789, Y 48.6039, Z -6.3333, A 0.000, B 0.000, C 0.000 }
gfCNCPoint5[3499] = {X 430.0204, Y 48.1273, Z -6.3333, A 0.000, B 0.000, C 0.000 }
gfCNCPoint5[3500] = {X 429.3871, Y 47.4940, Z -6.3333, A 0.000, B 0.000, C 0.000 }
gfCNCPoint5[3501] = {X 428.9105, Y 46.7355, Z -6.3333, A 0.000, B 0.000, C 0.000 }
gfCNCPoint5[3502] = {X 428.6147, Y 45.8901, Z -6.3333, A 0.000, B 0.000, C 0.000 }
gfCNCPoint5[3503] = {X 428.5144, Y 45.0000, Z -6.3333, A 0.000, B 0.000, C 0.000 }
gfCNCPoint5[3504] = {X 428.5148, Y 44.1538, Z -6.3333, A 0.000, B 0.000, C 0.000 }
gfCNCPoint5[3505] = {X 428.6096, Y 43.3414, Z -6.3333, A 0.000, B 0.000, C 0.000 }
gfCNCPoint5[3506] = {X 428.8676, Y 42.5654, Z -6.3333, A 0.000, B 0.000, C 0.000 }
gfCNCPoint5[3507] = {X 429.2781, Y 41.8580, Z -6.3333, A 0.000, B 0.000, C 0.000 }
gfCNCPoint5[3508] = {X 429.8239, Y 41.2489, Z -6.3333, A 0.000, B 0.000, C 0.000 }
gfCNCPoint5[3509] = {X 430.4821, Y 40.7635, Z -6.3333, A 0.000, B 0.000, C 0.000 }
gfCNCPoint5[3510] = {X 431.2253, Y 40.4222, Z -6.3333, A 0.000, B 0.000, C 0.000 }
gfCNCPoint5[3511] = {X 435.4112, Y 32.2288, Z -6.3333, A 0.000, B 0.000, C 0.000 }
gfCNCPoint5[3512] = {X 434.2188, Y 31.4711, Z -6.3333, A 0.000, B 0.000, C 0.000 }
gfCNCPoint5[3513] = {X 433.1334, Y 30.5667, Z -6.3333, A 0.000, B 0.000, C 0.000 }
gfCNCPoint5[3514] = {X 432.1728, Y 29.5307, Z -6.3333, A 0.000, B 0.000, C 0.000 }
gfCNCPoint5[3515] = {X 431.3530, Y 28.3801, Z -6.3333, A 0.000, B 0.000, C 0.000 }
gfCNCPoint5[3516] = {X 430.6874, Y 27.1339, Z -6.3333, A 0.000, B 0.000, C 0.000 }
gfCNCPoint5[3517] = {X 430.1870, Y 25.8127, Z -6.3333, A 0.000, B 0.000, C 0.000 }
gfCNCPoint5[3518] = {X 429.7648, Y 24.0028, Z -6.3333, A 0.000, B 0.000, C 0.000 }
gfCNCPoint5[3519] = {X 429.5522, Y 22.1565, Z -6.3333, A 0.000, B 0.000, C 0.000 }
gfCNCPoint5[3520] = {X 429.5522, Y 20.2980, Z -6.3333, A 0.000, B 0.000, C 0.000 }
gfCNCPoint5[3521] = {X 429.7648, Y 18.4516, Z -6.3333, A 0.000, B 0.000, C 0.000 }
gfCNCPoint5[3522] = {X 430.1870, Y 16.6417, Z -6.3333, A 0.000, B 0.000, C 0.000 }
gfCNCPoint5[3523] = {X 430.7414, Y 15.1518, Z -6.3333, A 0.000, B 0.000, C 0.000 }
gfCNCPoint5[3524] = {X 431.4958, Y 13.7526, Z -6.3333, A 0.000, B 0.000, C 0.000 }
gfCNCPoint5[3525] = {X 432.4358, Y 12.4706, Z -6.3333, A 0.000, B 0.000, C 0.000 }
gfCNCPoint5[3526] = {X 433.5435, Y 11.3304, Z -6.3333, A 0.000, B 0.000, C 0.000 }
gfCNCPoint5[3527] = {X 434.7977, Y 10.3537, Z -6.3333, A 0.000, B 0.000, C 0.000 }
gfCNCPoint5[3528] = {X 436.1746, Y 9.5591, Z -6.3333, A 0.000, B 0.000, C 0.000 }
gfCNCPoint5[3529] = {X 437.6478, Y 8.9618, Z -6.3333, A 0.000, B 0.000, C 0.000 }
gfCNCPoint5[3530] = {X 439.1893, Y 8.5732, Z -6.3333, A 0.000, B 0.000, C 0.000 }
gfCNCPoint5[3531] = {X 441.2579, Y 8.2867, Z -6.3333, A 0.000, B 0.000, C 0.000 }
gfCNCPoint5[3532] = {X 443.3442, Y 8.1940, Z -6.3333, A 0.000, B 0.000, C 0.000 }
gfCNCPoint5[3533] = {X 444.0367, Y 8.1899, Z -6.3333, A 0.000, B 0.000, C 0.000 }
gfCNCPoint5[3534] = {X 459.4468, Y 8.1899, Z -6.3333, A 0.000, B 0.000, C 0.000 }
gfCNCPoint5[3535] = {X 460.3349, Y 8.2900, Z -6.3333, A 0.000, B 0.000, C 0.000 }
gfCNCPoint5[3536] = {X 461.1785, Y 8.5851, Z -6.3333, A 0.000, B 0.000, C 0.000 }
gfCNCPoint5[3537] = {X 461.9352, Y 9.0606, Z -6.3333, A 0.000, B 0.000, C 0.000 }
gfCNCPoint5[3538] = {X 462.5672, Y 9.6926, Z -6.3333, A 0.000, B 0.000, C 0.000 }
gfCNCPoint5[3539] = {X 463.0427, Y 10.4493, Z -6.3333, A 0.000, B 0.000, C 0.000 }
gfCNCPoint5[3540] = {X 463.3379, Y 11.2929, Z -6.3333, A 0.000, B 0.000, C 0.000 }
gfCNCPoint5[3541] = {X 463.4379, Y 12.1810, Z -6.3333, A 0.000, B 0.000, C 0.000 }
gfCNCPoint5[3542] = {X 463.4378, Y 13.0163, Z -6.3333, A 0.000, B 0.000, C 0.000 }
gfCNCPoint5[3543] = {X 463.3398, Y 13.8587, Z -6.3333, A 0.000, B 0.000, C 0.000 }
gfCNCPoint5[3544] = {X 463.0664, Y 14.6616, Z -6.3333, A 0.000, B 0.000, C 0.000 }
gfCNCPoint5[3545] = {X 462.6299, Y 15.3887, Z -6.3333, A 0.000, B 0.000, C 0.000 }
gfCNCPoint5[3546] = {X 462.0499, Y 16.0075, Z -6.3333, A 0.000, B 0.000, C 0.000 }
gfCNCPoint5[3547] = {X 461.9728, Y 16.0723, Z -6.3333, A 0.000, B 0.000, C 0.000 }
gfCNCPoint5[3548] = {X 461.8942, Y 16.1351, Z -6.3333, A 0.000, B 0.000, C 0.000 }
gfCNCPoint5[3549] = {X 461.9112, Y 16.1933, Z -6.3333, A 0.000, B 0.000, C 0.000 }
gfCNCPoint5[3550] = {X 461.9106, Y 16.7687, Z -6.3333, A 0.000, B 0.000, C 0.000 }
gfCNCPoint5[3551] = {X 461.9111, Y 28.5935, Z -6.3333, A 0.000, B 0.000, C 0.000 }
gfCNCPoint5[3552] = {X 465.9914, Y 28.5933, Z -6.3333, A 0.000, B 0.000, C 0.000 }
gfCNCPoint5[3553] = {X 465.9914, Y 28.5933, Z -3.3333, A 0.000, B 0.000, C 0.000 }
gfCNCPoint5[3554] = {X 465.9914, Y 28.5933, Z 11.0000, A 0.000, B 0.000, C 0.000 }
gfCNCPoint5[3555] = {X 492.3835, Y 3.7899, Z 11.0000, A 0.000, B 0.000, C 0.000 }
gfCNCPoint5[3556] = {X 492.3835, Y 3.7899, Z -3.3333, A 0.000, B 0.000, C 0.000 }
gfCNCPoint5[3557] = {X 492.3835, Y 3.7899, Z -6.3333, A 0.000, B 0.000, C 0.000 }
gfCNCPoint5[3558] = {X 492.3835, Y 7.8699, Z -6.3333, A 0.000, B 0.000, C 0.000 }
gfCNCPoint5[3559] = {X 502.2066, Y 7.8699, Z -6.3333, A 0.000, B 0.000, C 0.000 }
gfCNCPoint5[3560] = {X 502.7395, Y 7.8741, Z -6.3333, A 0.000, B 0.000, C 0.000 }
gfCNCPoint5[3561] = {X 503.6914, Y 7.9883, Z -6.3333, A 0.000, B 0.000, C 0.000 }
gfCNCPoint5[3562] = {X 504.5943, Y 8.3105, Z -6.3333, A 0.000, B 0.000, C 0.000 }
gfCNCPoint5[3563] = {X 505.4035, Y 8.8246, Z -6.3333, A 0.000, B 0.000, C 0.000 }
gfCNCPoint5[3564] = {X 506.0788, Y 9.5052, Z -6.3333, A 0.000, B 0.000, C 0.000 }
gfCNCPoint5[3565] = {X 506.5866, Y 10.3184, Z -6.3333, A 0.000, B 0.000, C 0.000 }
gfCNCPoint5[3566] = {X 506.9017, Y 11.2238, Z -6.3333, A 0.000, B 0.000, C 0.000 }
gfCNCPoint5[3567] = {X 507.0085, Y 12.1765, Z -6.3333, A 0.000, B 0.000, C 0.000 }
gfCNCPoint5[3568] = {X 507.0085, Y 12.9782, Z -6.3333, A 0.000, B 0.000, C 0.000 }
gfCNCPoint5[3569] = {X 506.9072, Y 13.9079, Z -6.3333, A 0.000, B 0.000, C 0.000 }
gfCNCPoint5[3570] = {X 506.6082, Y 14.7940, Z -6.3333, A 0.000, B 0.000, C 0.000 }
gfCNCPoint5[3571] = {X 506.1256, Y 15.5951, Z -6.3333, A 0.000, B 0.000, C 0.000 }
gfCNCPoint5[3572] = {X 505.4818, Y 16.2734, Z -6.3333, A 0.000, B 0.000, C 0.000 }
gfCNCPoint5[3573] = {X 505.4817, Y 40.9133, Z -6.3333, A 0.000, B 0.000, C 0.000 }
gfCNCPoint5[3574] = {X 506.1199, Y 41.5843, Z -6.3333, A 0.000, B 0.000, C 0.000 }
gfCNCPoint5[3575] = {X 506.6004, Y 42.3758, Z -6.3333, A 0.000, B 0.000, C 0.000 }
gfCNCPoint5[3576] = {X 506.9011, Y 43.2516, Z -6.3333, A 0.000, B 0.000, C 0.000 }
gfCNCPoint5[3577] = {X 507.0083, Y 44.1713, Z -6.3333, A 0.000, B 0.000, C 0.000 }
gfCNCPoint5[3578] = {X 507.0085, Y 45.0000, Z -6.3333, A 0.000, B 0.000, C 0.000 }
gfCNCPoint5[3579] = {X 506.9002, Y 45.9613, Z -6.3333, A 0.000, B 0.000, C 0.000 }
gfCNCPoint5[3580] = {X 506.5807, Y 46.8744, Z -6.3333, A 0.000, B 0.000, C 0.000 }
gfCNCPoint5[3581] = {X 506.0660, Y 47.6935, Z -6.3333, A 0.000, B 0.000, C 0.000 }
gfCNCPoint5[3582] = {X 505.3820, Y 48.3775, Z -6.3333, A 0.000, B 0.000, C 0.000 }
gfCNCPoint5[3583] = {X 504.5629, Y 48.8922, Z -6.3333, A 0.000, B 0.000, C 0.000 }
gfCNCPoint5[3584] = {X 503.6498, Y 49.2117, Z -6.3333, A 0.000, B 0.000, C 0.000 }
gfCNCPoint5[3585] = {X 502.6885, Y 49.3200, Z -6.3333, A 0.000, B 0.000, C 0.000 }
gfCNCPoint5[3586] = {X 496.2450, Y 49.3200, Z -6.3333, A 0.000, B 0.000, C 0.000 }
gfCNCPoint5[3587] = {X 495.2885, Y 49.2128, Z -6.3333, A 0.000, B 0.000, C 0.000 }
gfCNCPoint5[3588] = {X 494.3794, Y 48.8964, Z -6.3333, A 0.000, B 0.000, C 0.000 }
gfCNCPoint5[3589] = {X 493.5630, Y 48.3866, Z -6.3333, A 0.000, B 0.000, C 0.000 }
gfCNCPoint5[3590] = {X 492.8797, Y 47.7087, Z -6.3333, A 0.000, B 0.000, C 0.000 }
gfCNCPoint5[3591] = {X 492.3635, Y 46.8963, Z -6.3333, A 0.000, B 0.000, C 0.000 }
gfCNCPoint5[3592] = {X 492.0399, Y 45.9898, Z -6.3333, A 0.000, B 0.000, C 0.000 }
gfCNCPoint5[3593] = {X 491.9252, Y 45.0341, Z -6.3333, A 0.000, B 0.000, C 0.000 }
gfCNCPoint5[3594] = {X 491.9254, Y 44.1494, Z -6.3333, A 0.000, B 0.000, C 0.000 }
gfCNCPoint5[3595] = {X 492.0359, Y 43.2364, Z -6.3333, A 0.000, B 0.000, C 0.000 }
gfCNCPoint5[3596] = {X 492.3371, Y 42.3675, Z -6.3333, A 0.000, B 0.000, C 0.000 }
gfCNCPoint5[3597] = {X 492.8153, Y 41.5821, Z -6.3333, A 0.000, B 0.000, C 0.000 }
gfCNCPoint5[3598] = {X 493.4490, Y 40.9157, Z -6.3333, A 0.000, B 0.000, C 0.000 }
gfCNCPoint5[3599] = {X 493.4490, Y 34.4738, Z -6.3333, A 0.000, B 0.000, C 0.000 }
gfCNCPoint5[3600] = {X 490.7251, Y 34.4738, Z -6.3333, A 0.000, B 0.000, C 0.000 }
gfCNCPoint5[3601] = {X 486.4405, Y 42.8175, Z -6.3333, A 0.000, B 0.000, C 0.000 }
gfCNCPoint5[3602] = {X 486.4452, Y 42.8305, Z -6.3333, A 0.000, B 0.000, C 0.000 }
gfCNCPoint5[3603] = {X 486.6110, Y 43.4913, Z -6.3333, A 0.000, B 0.000, C 0.000 }
gfCNCPoint5[3604] = {X 486.6708, Y 44.1699, Z -6.3333, A 0.000, B 0.000, C 0.000 }
gfCNCPoint5[3605] = {X 486.6710, Y 45.0000, Z -6.3333, A 0.000, B 0.000, C 0.000 }
gfCNCPoint5[3606] = {X 486.5627, Y 45.9613, Z -6.3333, A 0.000, B 0.000, C 0.000 }
gfCNCPoint5[3607] = {X 486.2432, Y 46.8744, Z -6.3333, A 0.000, B 0.000, C 0.000 }
gfCNCPoint5[3608] = {X 485.7285, Y 47.6935, Z -6.3333, A 0.000, B 0.000, C 0.000 }
gfCNCPoint5[3609] = {X 485.0445, Y 48.3775, Z -6.3333, A 0.000, B 0.000, C 0.000 }
gfCNCPoint5[3610] = {X 484.2254, Y 48.8922, Z -6.3333, A 0.000, B 0.000, C 0.000 }
gfCNCPoint5[3611] = {X 483.3123, Y 49.2117, Z -6.3333, A 0.000, B 0.000, C 0.000 }
gfCNCPoint5[3612] = {X 482.3510, Y 49.3200, Z -6.3333, A 0.000, B 0.000, C 0.000 }
gfCNCPoint5[3613] = {X 475.7650, Y 49.3200, Z -6.3333, A 0.000, B 0.000, C 0.000 }
gfCNCPoint5[3614] = {X 474.8037, Y 49.2117, Z -6.3333, A 0.000, B 0.000, C 0.000 }
gfCNCPoint5[3615] = {X 473.8906, Y 48.8922, Z -6.3333, A 0.000, B 0.000, C 0.000 }
gfCNCPoint5[3616] = {X 473.0715, Y 48.3775, Z -6.3333, A 0.000, B 0.000, C 0.000 }
gfCNCPoint5[3617] = {X 472.3875, Y 47.6935, Z -6.3333, A 0.000, B 0.000, C 0.000 }
gfCNCPoint5[3618] = {X 471.8728, Y 46.8745, Z -6.3333, A 0.000, B 0.000, C 0.000 }
gfCNCPoint5[3619] = {X 471.5533, Y 45.9614, Z -6.3333, A 0.000, B 0.000, C 0.000 }
gfCNCPoint5[3620] = {X 471.4450, Y 45.0001, Z -6.3333, A 0.000, B 0.000, C 0.000 }
gfCNCPoint5[3621] = {X 471.4454, Y 44.1494, Z -6.3333, A 0.000, B 0.000, C 0.000 }
gfCNCPoint5[3622] = {X 471.5430, Y 43.2935, Z -6.3333, A 0.000, B 0.000, C 0.000 }
gfCNCPoint5[3623] = {X 471.8086, Y 42.4740, Z -6.3333, A 0.000, B 0.000, C 0.000 }
gfCNCPoint5[3624] = {X 472.2314, Y 41.7236, Z -6.3333, A 0.000, B 0.000, C 0.000 }
gfCNCPoint5[3625] = {X 472.7947, Y 41.0719, Z -6.3333, A 0.000, B 0.000, C 0.000 }
gfCNCPoint5[3626] = {X 473.4762, Y 40.5449, Z -6.3333, A 0.000, B 0.000, C 0.000 }
gfCNCPoint5[3627] = {X 474.2486, Y 40.1637, Z -6.3333, A 0.000, B 0.000, C 0.000 }
